DATA_BLOCK "InstProfinetDeviceDiag_x2"   // DB209
AUTHOR : Siemens Digital Industries
FAMILY : LAF
VERSION : 1.2
// stored: AssignedProDiagFB ProDiag, InstanceOfName LAF_ProfinetDevDiag, InstanceOfType FB
"LAF_ProfinetDevDiag"
   // VAR_INPUT
   //    plantIdentifier { ExternalAccessible := 'False'; ExternalVisible := 'False'; ExternalWritable := 'False'} : WString[24] := WSTRING#'';
   //    textListId { ExternalAccessible := 'False'; ExternalVisible := 'False'; ExternalWritable := 'False'} : Int := 0;
   //    localProfinetSystem { ExternalAccessible := 'False'; ExternalVisible := 'False'; ExternalWritable := 'False'} : HW_IOSYSTEM := 0;
   //    firstCycle { ExternalAccessible := 'False'; ExternalVisible := 'False'; ExternalWritable := 'False'} : Bool := FALSE;
   //    maxDevicesDiag { ExternalAccessible := 'False'; ExternalVisible := 'False'; ExternalWritable := 'False'} : DInt := 0;
   //    maxModulesDiag { ExternalAccessible := 'False'; ExternalVisible := 'False'; ExternalWritable := 'False'} : DInt := 0;
   //    ackAlarms { ExternalAccessible := 'False'; ExternalVisible := 'False'; ExternalWritable := 'False'} : Bool := FALSE;
   //    hideAlarmMask { ExternalAccessible := 'False'; ExternalVisible := 'False'; ExternalWritable := 'False'} : Word := 16#0000;
   // END_VAR
   // VAR_OUTPUT
   //    generalAlarm { ExternalAccessible := 'False'; ExternalVisible := 'False'; ExternalWritable := 'False'} : Bool := FALSE;
   //    deviceFaulty { ExternalAccessible := 'False'; ExternalVisible := 'False'; ExternalWritable := 'False'} : Bool := FALSE;
   //    deviceProblem { ExternalAccessible := 'False'; ExternalVisible := 'False'; ExternalWritable := 'False'} : Bool := FALSE;
   //    deviceDeactivated { ExternalAccessible := 'False'; ExternalVisible := 'False'; ExternalWritable := 'False'} : Bool := FALSE;
   //    deviceNotPresent { ExternalAccessible := 'False'; ExternalVisible := 'False'; ExternalWritable := 'False'} : Bool := FALSE;
   // END_VAR
   // VAR_IN_OUT
   //    interfaceDevDiag : "LAF_typeDevDiagInterface";
   // END_VAR
   // VAR
   //    statDevDiagInternal { ExternalAccessible := 'False'; ExternalVisible := 'False'; ExternalWritable := 'False'} : "LAF_typeDevDiagInternal";
   //    statCnt1ShotGetName { ExternalAccessible := 'False'; ExternalVisible := 'False'; ExternalWritable := 'False'} : DInt := 1;
   //    statCnt1ShotGeo2Log { ExternalAccessible := 'False'; ExternalVisible := 'False'; ExternalWritable := 'False'} : DInt := 1;
   //    statCnt1ShotGetImDat { ExternalAccessible := 'False'; ExternalVisible := 'False'; ExternalWritable := 'False'} : DInt := 1;
   //    statCntCyclDevState { ExternalAccessible := 'False'; ExternalVisible := 'False'; ExternalWritable := 'False'} : DInt := 1;
   //    statCntCyclState { ExternalAccessible := 'False'; ExternalVisible := 'False'; ExternalWritable := 'False'} : DInt := 1;
   //    statCntCyclModulState { ExternalAccessible := 'False'; ExternalVisible := 'False'; ExternalWritable := 'False'} : DInt := 1;
   //    statCntCyclGetDiag { ExternalAccessible := 'False'; ExternalVisible := 'False'; ExternalWritable := 'False'} : DInt := 1;
   //    statBusy { ExternalAccessible := 'False'; ExternalVisible := 'False'; ExternalWritable := 'False'} : "LAF_typeDevDiagStateInstruct";
   //    statDone { ExternalAccessible := 'False'; ExternalVisible := 'False'; ExternalWritable := 'False'} : "LAF_typeDevDiagStateInstruct";
   //    statOtherInstruct { ExternalAccessible := 'False'; ExternalVisible := 'False'; ExternalWritable := 'False'} : "LAF_typeDevDiagInstruct";
   //    instGetName { ExternalAccessible := 'False'; ExternalVisible := 'False'; ExternalWritable := 'False'} : Get_Name;
   //    statGetNameDat { ExternalAccessible := 'False'; ExternalVisible := 'False'; ExternalWritable := 'False'} : String[24] := '';
   //    statGetNameErrorStatus { ExternalAccessible := 'False'; ExternalVisible := 'False'; ExternalWritable := 'False'} : Word := 16#0000;
   //    statGetNameErrorDevCycle { ExternalAccessible := 'False'; ExternalVisible := 'False'; ExternalWritable := 'False'} : DInt := 0;
   //    instGetImData { ExternalAccessible := 'False'; ExternalVisible := 'False'; ExternalWritable := 'False'} : Get_IM_Data;
   //    statIm0Data { ExternalAccessible := 'False'; ExternalVisible := 'False'; ExternalWritable := 'False'} : IM0_Data;
   //    statGetImDatErrorStatus { ExternalAccessible := 'False'; ExternalVisible := 'False'; ExternalWritable := 'False'} : Word := 16#0000;
   //    statGetImDatErrorCycle { ExternalAccessible := 'False'; ExternalVisible := 'False'; ExternalWritable := 'False'} : DInt := 0;
   //    statAlarm { ExternalAccessible := 'False'; ExternalVisible := 'False'; ExternalWritable := 'False'} : "LAF_typeDevDiagAlarm";
   //    statHideAlarm { ExternalAccessible := 'False'; ExternalVisible := 'False'; ExternalWritable := 'False'} : "LAF_typeDevDiagAlarm";
   //    statRisPushbutton { ExternalAccessible := 'False'; ExternalVisible := 'False'; ExternalWritable := 'False'} : "LAF_typeDevDiagRisEdge";
   //    statErrorText { ExternalAccessible := 'False'; ExternalVisible := 'False'; ExternalWritable := 'False'} : String[24] := 'No Device Name readable';
   //    stat8CharError { ExternalAccessible := 'False'; ExternalVisible := 'False'; ExternalWritable := 'False'} : String[8] := '????????';
   //    statAlarmNo { ExternalAccessible := 'False'; ExternalVisible := 'False'; ExternalWritable := 'False'} : Array[0..23] of UInt;
   // END_VAR
BEGIN
   statDevDiagInternal.localProfinetSystem := 0;
   statDevDiagInternal.maxDevices := 0;
   statDevDiagInternal.maxModules := 0;
   statDevDiagInternal.numberDevices.configured := 0;
   statDevDiagInternal.numberDevices.notPresent := 0;
   statDevDiagInternal.numberDevices.deactivated := 0;
   statDevDiagInternal.numberDevices.faulty := 0;
   statDevDiagInternal.numberDevices.problem := 0;
   statDevDiagInternal.hwAddress[0..256].hwtype2 := 0;
   statDevDiagInternal.hwAddress[0..256].hwtype5 := 0;
   statDevDiagInternal.hwAddress[0..256].hwtype5If := 0;
   statBusy.getName := FALSE;
   statBusy.geo2Log := FALSE;
   statBusy.moduleStates := FALSE;
   statBusy.getDiag := FALSE;
   statBusy.getImData := FALSE;
   statDone.getName := FALSE;
   statDone.geo2Log := FALSE;
   statDone.moduleStates := FALSE;
   statDone.getDiag := FALSE;
   statDone.getImData := FALSE;
   statOtherInstruct.log2GeoLaddr := 0;
   statOtherInstruct.log2GeoRetVal := 0;
   statOtherInstruct.log2Geo.HWTYPE := 0;
   statOtherInstruct.log2Geo.AREA := 0;
   statOtherInstruct.log2Geo.IOSYSTEM := 0;
   statOtherInstruct.log2Geo.STATION := 0;
   statOtherInstruct.log2Geo.SLOT := 0;
   statOtherInstruct.log2Geo.SUBSLOT := 0;
   statOtherInstruct.devStateMode1.laddr := 0;
   statOtherInstruct.devStateMode1.mode := 0;
   statOtherInstruct.devStateMode1.retVal := 0;
   statOtherInstruct.devStateMode1.state[0..1024] := FALSE;
   statOtherInstruct.devStateMode2.laddr := 0;
   statOtherInstruct.devStateMode2.mode := 0;
   statOtherInstruct.devStateMode2.retVal := 0;
   statOtherInstruct.devStateMode2.state[0..1024] := FALSE;
   statOtherInstruct.devStateMode3.laddr := 0;
   statOtherInstruct.devStateMode3.mode := 0;
   statOtherInstruct.devStateMode3.retVal := 0;
   statOtherInstruct.devStateMode3.state[0..1024] := FALSE;
   statOtherInstruct.devStateMode4.laddr := 0;
   statOtherInstruct.devStateMode4.mode := 0;
   statOtherInstruct.devStateMode4.retVal := 0;
   statOtherInstruct.devStateMode4.state[0..1024] := FALSE;
   statOtherInstruct.devStateMode5.laddr := 0;
   statOtherInstruct.devStateMode5.mode := 0;
   statOtherInstruct.devStateMode5.retVal := 0;
   statOtherInstruct.devStateMode5.state[0..1024] := FALSE;
   statOtherInstruct.geo2LogLaddr := 0;
   statOtherInstruct.geo2LogRetVal := 0;
   statOtherInstruct.geo2Log.HWTYPE := 0;
   statOtherInstruct.geo2Log.AREA := 0;
   statOtherInstruct.geo2Log.IOSYSTEM := 0;
   statOtherInstruct.geo2Log.STATION := 0;
   statOtherInstruct.geo2Log.SLOT := 0;
   statOtherInstruct.geo2Log.SUBSLOT := 0;
   statOtherInstruct.moduleStateMode2.laddr := 0;
   statOtherInstruct.moduleStateMode2.mode := 0;
   statOtherInstruct.moduleStateMode2.retVal := 0;
   statOtherInstruct.moduleStateMode2.state[0..127] := FALSE;
   statOtherInstruct.moduleStateMode5.laddr := 0;
   statOtherInstruct.moduleStateMode5.mode := 0;
   statOtherInstruct.moduleStateMode5.retVal := 0;
   statOtherInstruct.moduleStateMode5.state[0..127] := FALSE;
   statOtherInstruct.getDiag.mode := 0;
   statOtherInstruct.getDiag.laddr := 0;
   statOtherInstruct.getDiag.retVal := 0;
   statOtherInstruct.getDiag.cntDiag := 0;
   statOtherInstruct.getDiag.diagDataMode0 := 16#0000_0000;
   statOtherInstruct.getDiag.diagDataMode1.MaintainanceState := 16#0000_0000;
   statOtherInstruct.getDiag.diagDataMode1.ComponentStateDetail := 16#0000_0000;
   statOtherInstruct.getDiag.diagDataMode1.OwnState := 0;
   statOtherInstruct.getDiag.diagDataMode1.IOState := 16#0000;
   statOtherInstruct.getDiag.diagDataMode1.OperatingState := 0;
   statOtherInstruct.getDiag.diagDataMode2.SubordinateState := 0;
   statOtherInstruct.getDiag.diagDataMode2.SubordinateIOState := 16#0000;
   statOtherInstruct.getDiag.diagDataMode2.DNNmode := 16#0000;
   statOtherInstruct.getDiag.detailData := 0;
   instGetName.LADDR := 0;
   instGetName.STATION_NR := 0;
   instGetName.DONE := FALSE;
   instGetName.BUSY := FALSE;
   instGetName.ERROR := FALSE;
   instGetName.LEN := 0;
   instGetName.STATUS := 16#0000;
   instGetName.BusyState := 16#0000;
   instGetImData.LADDR := 0;
   instGetImData.IM_TYPE := 0;
   instGetImData.DONE := FALSE;
   instGetImData.BUSY := FALSE;
   instGetImData.ERROR := FALSE;
   instGetImData.STATUS := 16#0000;
   instGetImData.sdw_GetAttrID := 16#0000_0000;
   instGetImData.sdw_GetAttrAID := 16#0000_0000;
   instGetImData.sdi_SfcLen := 0;
   instGetImData.sb_useGetMultiAttr := FALSE;
   instGetImData.sui_GetMultiAttrACount := 0;
   instGetImData.sa_GetMultiAttrPathLens[0] := 0;
   instGetImData.sa_GetMultiAttrPaths[0..2] := 0;
   instGetImData.sa_GetMultiAttrResultLens[0] := 0;
   instGetImData.sa_GetMultiAttrResult := '';
   instGetImData.sb_SfcValid := FALSE;
   instGetImData.sb_SfcERROR := FALSE;
   instGetImData.sw_SfcStatus := 16#0000;
   instGetImData.sa_SfcData[0..64] := 16#00;
   instGetImData.sudi_arraylength := 0;
   instGetImData.sudi_datatype := 0;
   instGetImData.sui_imdataLen := 0;
   instGetImData.sui_imdataLen_netto := 54;
   instGetImData.si_index := 0;
   instGetImData.sb_SfcLocked := FALSE;
   instGetImData.pw_TemporaryWord := 16#0000;
   instGetImData.pa_DataByte[0..53] := 16#00;
   instGetImData.pa_DataChar[0..53] := ' ';
   instGetImData.pa_TemporaryCharArray[0..19] := ' ';
   instGetImData.p_DataUDT.Manufacturer_ID := 0;
   instGetImData.p_DataUDT.Order_ID := '';
   instGetImData.p_DataUDT.Serial_Number := '';
   instGetImData.p_DataUDT.Hardware_Revision := 0;
   instGetImData.p_DataUDT.Software_Revision."Type" := ' ';
   instGetImData.p_DataUDT.Software_Revision.Functional := 0;
   instGetImData.p_DataUDT.Software_Revision.Bugfix := 0;
   instGetImData.p_DataUDT.Software_Revision.Internal := 0;
   instGetImData.p_DataUDT.Revision_Counter := 0;
   instGetImData.p_DataUDT.Profile_ID := 0;
   instGetImData.p_DataUDT.Profile_Specific_Type := 0;
   instGetImData.p_DataUDT.IM_Version := 16#0000;
   instGetImData.p_DataUDT.IM_Supported := 16#0000;
   statIm0Data.Manufacturer_ID := 0;
   statIm0Data.Order_ID := '';
   statIm0Data.Serial_Number := '';
   statIm0Data.Hardware_Revision := 0;
   statIm0Data.Software_Revision."Type" := ' ';
   statIm0Data.Software_Revision.Functional := 0;
   statIm0Data.Software_Revision.Bugfix := 0;
   statIm0Data.Software_Revision.Internal := 0;
   statIm0Data.Revision_Counter := 0;
   statIm0Data.Profile_ID := 0;
   statIm0Data.Profile_Specific_Type := 0;
   statIm0Data.IM_Version := 16#0000;
   statIm0Data.IM_Supported := 16#0000;
   statAlarm.invalidValueMaxDevices := FALSE;
   statAlarm.invalidValueMaxModules := FALSE;
   statAlarm.invalidAddressLog2Geo := FALSE;
   statAlarm.errorReadDeviceStates := FALSE;
   statAlarm.deviceFaulty := FALSE;
   statAlarm.deviceProblem := FALSE;
   statAlarm.deviceDeactivated := FALSE;
   statAlarm.deviceNotPresent := FALSE;
   statAlarm.deviceNetworkError := FALSE;
   statAlarm.deviceMaintRequired := FALSE;
   statAlarm.deviceMaintDemanded := FALSE;
   statAlarm.spare11 := FALSE;
   statAlarm.spare12 := FALSE;
   statAlarm.spare13 := FALSE;
   statAlarm.spare14 := FALSE;
   statAlarm.spare15 := FALSE;
   statHideAlarm.invalidValueMaxDevices := FALSE;
   statHideAlarm.invalidValueMaxModules := FALSE;
   statHideAlarm.invalidAddressLog2Geo := FALSE;
   statHideAlarm.errorReadDeviceStates := FALSE;
   statHideAlarm.deviceFaulty := FALSE;
   statHideAlarm.deviceProblem := FALSE;
   statHideAlarm.deviceDeactivated := FALSE;
   statHideAlarm.deviceNotPresent := FALSE;
   statHideAlarm.deviceNetworkError := FALSE;
   statHideAlarm.deviceMaintRequired := FALSE;
   statHideAlarm.deviceMaintDemanded := FALSE;
   statHideAlarm.spare11 := FALSE;
   statHideAlarm.spare12 := FALSE;
   statHideAlarm.spare13 := FALSE;
   statHideAlarm.spare14 := FALSE;
   statHideAlarm.spare15 := FALSE;
   statRisPushbutton.risEdgeManualReadAll := FALSE;
   statRisPushbutton.posPulseManualReadAll := FALSE;
   statRisPushbutton.risEdgeResetAll := FALSE;
   statRisPushbutton.posPulseResetAll := FALSE;
   statRisPushbutton.risEdgeQuitAlarms := FALSE;
   statRisPushbutton.posPulseQuitAlarms := FALSE;
   statAlarmNo[0] := 0;
   statAlarmNo[1] := 1;
   statAlarmNo[2] := 2;
   statAlarmNo[3] := 3;
   statAlarmNo[4] := 4;
   statAlarmNo[5] := 5;
   statAlarmNo[6] := 6;
   statAlarmNo[7] := 7;
   statAlarmNo[8] := 8;
   statAlarmNo[9] := 9;
   statAlarmNo[10] := 10;
   statAlarmNo[11] := 11;
   statAlarmNo[12] := 12;
   statAlarmNo[13] := 13;
   statAlarmNo[14] := 14;
   statAlarmNo[15] := 15;
   statAlarmNo[16] := 16;
   statAlarmNo[17] := 17;
   statAlarmNo[18] := 18;
   statAlarmNo[19] := 19;
   statAlarmNo[20] := 20;
   statAlarmNo[21] := 21;
   statAlarmNo[22] := 22;
   statAlarmNo[23] := 23;
END_DATA_BLOCK

DATA_BLOCK "CallInterfaceSignalsConv_BA10"   // DB347
// stored: InstanceOfName CallInterfaceSignalsConv, InstanceOfType FB
"CallInterfaceSignalsConv"
BEGIN
   signalsS2R.Load_Enable := FALSE;
   signalsS2R.Load_Complete_Comfirm := FALSE;
   signalsS2R.Cell_Data_Report := FALSE;
   signalsS2R.signal3 := FALSE;
   signalsS2R.signal4 := FALSE;
   signalsS2R.signal5 := FALSE;
   signalsS2R.signal6 := FALSE;
   signalsS2R.signal7 := FALSE;
   signalsS2R.signal8 := FALSE;
   signalsS2R.signal9 := FALSE;
   signalsS2R.signal10 := FALSE;
   signalsS2R.signal11 := FALSE;
   signalsS2R.signal12 := FALSE;
   signalsS2R.signal13 := FALSE;
   signalsS2R.signal14 := FALSE;
   signalsS2R.HeartBeat := FALSE;
   signalsS2R.signal16 := FALSE;
   signalsS2R.signal17 := FALSE;
   signalsS2R.signal18 := FALSE;
   signalsS2R.signal19 := FALSE;
   signalsS2R.signal20 := FALSE;
   signalsS2R.signal21 := FALSE;
   signalsS2R.signal22 := FALSE;
   signalsS2R.signal23 := FALSE;
   signalsS2R.signal24 := FALSE;
   signalsS2R.signal25 := FALSE;
   signalsS2R.signal26 := FALSE;
   signalsS2R.signal27 := FALSE;
   signalsS2R.signal28 := FALSE;
   signalsS2R.signal29 := FALSE;
   signalsS2R.signal30 := FALSE;
   signalsS2R.signal31 := FALSE;
   signalsS2R.signal32 := FALSE;
   signalsS2R.signal33 := FALSE;
   signalsS2R.signal34 := FALSE;
   signalsS2R.signal35 := FALSE;
   signalsS2R.signal36 := FALSE;
   signalsS2R.signal37 := FALSE;
   signalsS2R.signal38 := FALSE;
   signalsS2R.signal39 := FALSE;
   signalsS2R.signal40 := FALSE;
   signalsS2R.signal41 := FALSE;
   signalsS2R.signal42 := FALSE;
   signalsS2R.signal43 := FALSE;
   signalsS2R.signal44 := FALSE;
   signalsS2R.signal45 := FALSE;
   signalsS2R.signal46 := FALSE;
   signalsS2R.signal47 := FALSE;
   signalsS2R.signal48 := FALSE;
   signalsS2R.signal49 := FALSE;
   signalsS2R.signal50 := FALSE;
   signalsS2R.signal51 := FALSE;
   signalsS2R.signal52 := FALSE;
   signalsS2R.signal53 := FALSE;
   signalsS2R.signal54 := FALSE;
   signalsS2R.signal55 := FALSE;
   signalsS2R.signal56 := FALSE;
   signalsS2R.signal57 := FALSE;
   signalsS2R.signal58 := FALSE;
   signalsS2R.signal59 := FALSE;
   signalsS2R.signal60 := FALSE;
   signalsS2R.signal61 := FALSE;
   signalsS2R.signal62 := FALSE;
   signalsS2R.signal63 := FALSE;
   signalsS2R.signal64 := FALSE;
   signalsS2R.signal65 := FALSE;
   signalsS2R.signal66 := FALSE;
   signalsS2R.signal67 := FALSE;
   signalsS2R.signal68 := FALSE;
   signalsS2R.signal69 := FALSE;
   signalsS2R.signal70 := FALSE;
   signalsS2R.signal71 := FALSE;
   signalsS2R.signal72 := FALSE;
   signalsS2R.signal73 := FALSE;
   signalsS2R.signal74 := FALSE;
   signalsS2R.signal75 := FALSE;
   signalsS2R.signal76 := FALSE;
   signalsS2R.signal77 := FALSE;
   signalsS2R.signal78 := FALSE;
   signalsS2R.signal79 := FALSE;
   signalsS2R.signal80 := FALSE;
   signalsS2R.signal81 := FALSE;
   signalsS2R.signal82 := FALSE;
   signalsS2R.signal83 := FALSE;
   signalsS2R.signal84 := FALSE;
   signalsS2R.signal85 := FALSE;
   signalsS2R.signal86 := FALSE;
   signalsS2R.signal87 := FALSE;
   signalsS2R.signal88 := FALSE;
   signalsS2R.signal89 := FALSE;
   signalsS2R.signal90 := FALSE;
   signalsS2R.signal91 := FALSE;
   signalsS2R.signal92 := FALSE;
   signalsS2R.signal93 := FALSE;
   signalsS2R.signal94 := FALSE;
   signalsS2R.signal95 := FALSE;
   signalsR2S.Load_Requset := FALSE;
   signalsR2S.Load_Busy := FALSE;
   signalsR2S.Load_Complete := FALSE;
   signalsR2S.Cell_Data_Request := FALSE;
   signalsR2S.Cell_Data_Report_Ack := FALSE;
   signalsR2S.Cell_Data_Report_Nck := FALSE;
   signalsR2S.signal6 := FALSE;
   signalsR2S.signal7 := FALSE;
   signalsR2S.signal8 := FALSE;
   signalsR2S.signal9 := FALSE;
   signalsR2S.signal10 := FALSE;
   signalsR2S.signal11 := FALSE;
   signalsR2S.signal12 := FALSE;
   signalsR2S.signal13 := FALSE;
   signalsR2S.signal14 := FALSE;
   signalsR2S.HeartBeat := FALSE;
   signalsR2S.signal16 := FALSE;
   signalsR2S.signal17 := FALSE;
   signalsR2S.signal18 := FALSE;
   signalsR2S.signal19 := FALSE;
   signalsR2S.signal20 := FALSE;
   signalsR2S.signal21 := FALSE;
   signalsR2S.signal22 := FALSE;
   signalsR2S.signal23 := FALSE;
   signalsR2S.signal24 := FALSE;
   signalsR2S.signal25 := FALSE;
   signalsR2S.signal26 := FALSE;
   signalsR2S.signal27 := FALSE;
   signalsR2S.signal28 := FALSE;
   signalsR2S.signal29 := FALSE;
   signalsR2S.signal30 := FALSE;
   signalsR2S.signal31 := FALSE;
   signalsR2S.signal32 := FALSE;
   signalsR2S.signal33 := FALSE;
   signalsR2S.signal34 := FALSE;
   signalsR2S.signal35 := FALSE;
   signalsR2S.signal36 := FALSE;
   signalsR2S.signal37 := FALSE;
   signalsR2S.signal38 := FALSE;
   signalsR2S.signal39 := FALSE;
   signalsR2S.signal40 := FALSE;
   signalsR2S.signal41 := FALSE;
   signalsR2S.signal42 := FALSE;
   signalsR2S.signal43 := FALSE;
   signalsR2S.signal44 := FALSE;
   signalsR2S.signal45 := FALSE;
   signalsR2S.signal46 := FALSE;
   signalsR2S.signal47 := FALSE;
   signalsR2S.signal48 := FALSE;
   signalsR2S.signal49 := FALSE;
   signalsR2S.signal50 := FALSE;
   signalsR2S.signal51 := FALSE;
   signalsR2S.signal52 := FALSE;
   signalsR2S.signal53 := FALSE;
   signalsR2S.signal54 := FALSE;
   signalsR2S.signal55 := FALSE;
   signalsR2S.signal56 := FALSE;
   signalsR2S.signal57 := FALSE;
   signalsR2S.signal58 := FALSE;
   signalsR2S.signal59 := FALSE;
   signalsR2S.signal60 := FALSE;
   signalsR2S.signal61 := FALSE;
   signalsR2S.signal62 := FALSE;
   signalsR2S.signal63 := FALSE;
   signalsR2S.signal64 := FALSE;
   signalsR2S.signal65 := FALSE;
   signalsR2S.signal66 := FALSE;
   signalsR2S.signal67 := FALSE;
   signalsR2S.signal68 := FALSE;
   signalsR2S.signal69 := FALSE;
   signalsR2S.signal70 := FALSE;
   signalsR2S.signal71 := FALSE;
   signalsR2S.signal72 := FALSE;
   signalsR2S.signal73 := FALSE;
   signalsR2S.signal74 := FALSE;
   signalsR2S.signal75 := FALSE;
   signalsR2S.signal76 := FALSE;
   signalsR2S.signal77 := FALSE;
   signalsR2S.signal78 := FALSE;
   signalsR2S.signal79 := FALSE;
   signalsR2S.signal80 := FALSE;
   signalsR2S.signal81 := FALSE;
   signalsR2S.signal82 := FALSE;
   signalsR2S.signal83 := FALSE;
   signalsR2S.signal84 := FALSE;
   signalsR2S.signal85 := FALSE;
   signalsR2S.signal86 := FALSE;
   signalsR2S.signal87 := FALSE;
   signalsR2S.signal88 := FALSE;
   signalsR2S.signal89 := FALSE;
   signalsR2S.signal90 := FALSE;
   signalsR2S.signal91 := FALSE;
   signalsR2S.signal92 := FALSE;
   signalsR2S.signal93 := FALSE;
   signalsR2S.signal94 := FALSE;
   signalsR2S.signal95 := FALSE;
   statWordBuffer_2[0..5] := 16#0000;
   statWordBuffer_1[0..5] := 16#0000;
END_DATA_BLOCK

DATA_BLOCK "CallInterfaceSignalsConv_BA15"   // DB348
// stored: InstanceOfName CallInterfaceSignalsConv, InstanceOfType FB
"CallInterfaceSignalsConv"
BEGIN
   signalsS2R.Load_Enable := FALSE;
   signalsS2R.Load_Complete_Comfirm := FALSE;
   signalsS2R.Cell_Data_Report := FALSE;
   signalsS2R.signal3 := FALSE;
   signalsS2R.signal4 := FALSE;
   signalsS2R.signal5 := FALSE;
   signalsS2R.signal6 := FALSE;
   signalsS2R.signal7 := FALSE;
   signalsS2R.signal8 := FALSE;
   signalsS2R.signal9 := FALSE;
   signalsS2R.signal10 := FALSE;
   signalsS2R.signal11 := FALSE;
   signalsS2R.signal12 := FALSE;
   signalsS2R.signal13 := FALSE;
   signalsS2R.signal14 := FALSE;
   signalsS2R.HeartBeat := FALSE;
   signalsS2R.signal16 := FALSE;
   signalsS2R.signal17 := FALSE;
   signalsS2R.signal18 := FALSE;
   signalsS2R.signal19 := FALSE;
   signalsS2R.signal20 := FALSE;
   signalsS2R.signal21 := FALSE;
   signalsS2R.signal22 := FALSE;
   signalsS2R.signal23 := FALSE;
   signalsS2R.signal24 := FALSE;
   signalsS2R.signal25 := FALSE;
   signalsS2R.signal26 := FALSE;
   signalsS2R.signal27 := FALSE;
   signalsS2R.signal28 := FALSE;
   signalsS2R.signal29 := FALSE;
   signalsS2R.signal30 := FALSE;
   signalsS2R.signal31 := FALSE;
   signalsS2R.signal32 := FALSE;
   signalsS2R.signal33 := FALSE;
   signalsS2R.signal34 := FALSE;
   signalsS2R.signal35 := FALSE;
   signalsS2R.signal36 := FALSE;
   signalsS2R.signal37 := FALSE;
   signalsS2R.signal38 := FALSE;
   signalsS2R.signal39 := FALSE;
   signalsS2R.signal40 := FALSE;
   signalsS2R.signal41 := FALSE;
   signalsS2R.signal42 := FALSE;
   signalsS2R.signal43 := FALSE;
   signalsS2R.signal44 := FALSE;
   signalsS2R.signal45 := FALSE;
   signalsS2R.signal46 := FALSE;
   signalsS2R.signal47 := FALSE;
   signalsS2R.signal48 := FALSE;
   signalsS2R.signal49 := FALSE;
   signalsS2R.signal50 := FALSE;
   signalsS2R.signal51 := FALSE;
   signalsS2R.signal52 := FALSE;
   signalsS2R.signal53 := FALSE;
   signalsS2R.signal54 := FALSE;
   signalsS2R.signal55 := FALSE;
   signalsS2R.signal56 := FALSE;
   signalsS2R.signal57 := FALSE;
   signalsS2R.signal58 := FALSE;
   signalsS2R.signal59 := FALSE;
   signalsS2R.signal60 := FALSE;
   signalsS2R.signal61 := FALSE;
   signalsS2R.signal62 := FALSE;
   signalsS2R.signal63 := FALSE;
   signalsS2R.signal64 := FALSE;
   signalsS2R.signal65 := FALSE;
   signalsS2R.signal66 := FALSE;
   signalsS2R.signal67 := FALSE;
   signalsS2R.signal68 := FALSE;
   signalsS2R.signal69 := FALSE;
   signalsS2R.signal70 := FALSE;
   signalsS2R.signal71 := FALSE;
   signalsS2R.signal72 := FALSE;
   signalsS2R.signal73 := FALSE;
   signalsS2R.signal74 := FALSE;
   signalsS2R.signal75 := FALSE;
   signalsS2R.signal76 := FALSE;
   signalsS2R.signal77 := FALSE;
   signalsS2R.signal78 := FALSE;
   signalsS2R.signal79 := FALSE;
   signalsS2R.signal80 := FALSE;
   signalsS2R.signal81 := FALSE;
   signalsS2R.signal82 := FALSE;
   signalsS2R.signal83 := FALSE;
   signalsS2R.signal84 := FALSE;
   signalsS2R.signal85 := FALSE;
   signalsS2R.signal86 := FALSE;
   signalsS2R.signal87 := FALSE;
   signalsS2R.signal88 := FALSE;
   signalsS2R.signal89 := FALSE;
   signalsS2R.signal90 := FALSE;
   signalsS2R.signal91 := FALSE;
   signalsS2R.signal92 := FALSE;
   signalsS2R.signal93 := FALSE;
   signalsS2R.signal94 := FALSE;
   signalsS2R.signal95 := FALSE;
   signalsR2S.Load_Requset := FALSE;
   signalsR2S.Load_Busy := FALSE;
   signalsR2S.Load_Complete := FALSE;
   signalsR2S.Cell_Data_Request := FALSE;
   signalsR2S.Cell_Data_Report_Ack := FALSE;
   signalsR2S.Cell_Data_Report_Nck := FALSE;
   signalsR2S.signal6 := FALSE;
   signalsR2S.signal7 := FALSE;
   signalsR2S.signal8 := FALSE;
   signalsR2S.signal9 := FALSE;
   signalsR2S.signal10 := FALSE;
   signalsR2S.signal11 := FALSE;
   signalsR2S.signal12 := FALSE;
   signalsR2S.signal13 := FALSE;
   signalsR2S.signal14 := FALSE;
   signalsR2S.HeartBeat := FALSE;
   signalsR2S.signal16 := FALSE;
   signalsR2S.signal17 := FALSE;
   signalsR2S.signal18 := FALSE;
   signalsR2S.signal19 := FALSE;
   signalsR2S.signal20 := FALSE;
   signalsR2S.signal21 := FALSE;
   signalsR2S.signal22 := FALSE;
   signalsR2S.signal23 := FALSE;
   signalsR2S.signal24 := FALSE;
   signalsR2S.signal25 := FALSE;
   signalsR2S.signal26 := FALSE;
   signalsR2S.signal27 := FALSE;
   signalsR2S.signal28 := FALSE;
   signalsR2S.signal29 := FALSE;
   signalsR2S.signal30 := FALSE;
   signalsR2S.signal31 := FALSE;
   signalsR2S.signal32 := FALSE;
   signalsR2S.signal33 := FALSE;
   signalsR2S.signal34 := FALSE;
   signalsR2S.signal35 := FALSE;
   signalsR2S.signal36 := FALSE;
   signalsR2S.signal37 := FALSE;
   signalsR2S.signal38 := FALSE;
   signalsR2S.signal39 := FALSE;
   signalsR2S.signal40 := FALSE;
   signalsR2S.signal41 := FALSE;
   signalsR2S.signal42 := FALSE;
   signalsR2S.signal43 := FALSE;
   signalsR2S.signal44 := FALSE;
   signalsR2S.signal45 := FALSE;
   signalsR2S.signal46 := FALSE;
   signalsR2S.signal47 := FALSE;
   signalsR2S.signal48 := FALSE;
   signalsR2S.signal49 := FALSE;
   signalsR2S.signal50 := FALSE;
   signalsR2S.signal51 := FALSE;
   signalsR2S.signal52 := FALSE;
   signalsR2S.signal53 := FALSE;
   signalsR2S.signal54 := FALSE;
   signalsR2S.signal55 := FALSE;
   signalsR2S.signal56 := FALSE;
   signalsR2S.signal57 := FALSE;
   signalsR2S.signal58 := FALSE;
   signalsR2S.signal59 := FALSE;
   signalsR2S.signal60 := FALSE;
   signalsR2S.signal61 := FALSE;
   signalsR2S.signal62 := FALSE;
   signalsR2S.signal63 := FALSE;
   signalsR2S.signal64 := FALSE;
   signalsR2S.signal65 := FALSE;
   signalsR2S.signal66 := FALSE;
   signalsR2S.signal67 := FALSE;
   signalsR2S.signal68 := FALSE;
   signalsR2S.signal69 := FALSE;
   signalsR2S.signal70 := FALSE;
   signalsR2S.signal71 := FALSE;
   signalsR2S.signal72 := FALSE;
   signalsR2S.signal73 := FALSE;
   signalsR2S.signal74 := FALSE;
   signalsR2S.signal75 := FALSE;
   signalsR2S.signal76 := FALSE;
   signalsR2S.signal77 := FALSE;
   signalsR2S.signal78 := FALSE;
   signalsR2S.signal79 := FALSE;
   signalsR2S.signal80 := FALSE;
   signalsR2S.signal81 := FALSE;
   signalsR2S.signal82 := FALSE;
   signalsR2S.signal83 := FALSE;
   signalsR2S.signal84 := FALSE;
   signalsR2S.signal85 := FALSE;
   signalsR2S.signal86 := FALSE;
   signalsR2S.signal87 := FALSE;
   signalsR2S.signal88 := FALSE;
   signalsR2S.signal89 := FALSE;
   signalsR2S.signal90 := FALSE;
   signalsR2S.signal91 := FALSE;
   signalsR2S.signal92 := FALSE;
   signalsR2S.signal93 := FALSE;
   signalsR2S.signal94 := FALSE;
   signalsR2S.signal95 := FALSE;
   statWordBuffer_2[0..5] := 16#0000;
   statWordBuffer_1[0..5] := 16#0000;
END_DATA_BLOCK

DATA_BLOCK "InterfaceSignals"   // DB232
// stored: Access Published, InstanceOfName LER_SignalsInterface, InstanceOfType UDT
"LER_SignalsInterface"
   // VAR
   //    HMI_Select_Mode : Bool := FALSE;
   //    ButtonValue : Array[0..16] of "LER_SignalsInput";
   // END_VAR
BEGIN
   ButtonValue[0].ButtonLeft[0..15] := FALSE;
   ButtonValue[1].ButtonLeft[0..15] := FALSE;
   ButtonValue[2].ButtonLeft[0..15] := FALSE;
   ButtonValue[3].ButtonLeft[0..15] := FALSE;
   ButtonValue[4].ButtonLeft[0..15] := FALSE;
   ButtonValue[5].ButtonLeft[0..15] := FALSE;
   ButtonValue[6].ButtonLeft[0..15] := FALSE;
   ButtonValue[7].ButtonLeft[0..15] := FALSE;
   ButtonValue[8].ButtonLeft[0..15] := FALSE;
   ButtonValue[9].ButtonLeft[0..15] := FALSE;
   ButtonValue[10].ButtonLeft[0..15] := FALSE;
   ButtonValue[11].ButtonLeft[0..15] := FALSE;
   ButtonValue[12].ButtonLeft[0..15] := FALSE;
   ButtonValue[13].ButtonLeft[0..15] := FALSE;
   ButtonValue[14].ButtonLeft[0..15] := FALSE;
   ButtonValue[15].ButtonLeft[0..15] := FALSE;
   ButtonValue[16].ButtonLeft[0..15] := FALSE;
   ButtonValue[0].ButtonRight[0..15] := FALSE;
   ButtonValue[1].ButtonRight[0..15] := FALSE;
   ButtonValue[2].ButtonRight[0..15] := FALSE;
   ButtonValue[3].ButtonRight[0..15] := FALSE;
   ButtonValue[4].ButtonRight[0..15] := FALSE;
   ButtonValue[5].ButtonRight[0..15] := FALSE;
   ButtonValue[6].ButtonRight[0..15] := FALSE;
   ButtonValue[7].ButtonRight[0..15] := FALSE;
   ButtonValue[8].ButtonRight[0..15] := FALSE;
   ButtonValue[9].ButtonRight[0..15] := FALSE;
   ButtonValue[10].ButtonRight[0..15] := FALSE;
   ButtonValue[11].ButtonRight[0..15] := FALSE;
   ButtonValue[12].ButtonRight[0..15] := FALSE;
   ButtonValue[13].ButtonRight[0..15] := FALSE;
   ButtonValue[14].ButtonRight[0..15] := FALSE;
   ButtonValue[15].ButtonRight[0..15] := FALSE;
   ButtonValue[16].ButtonRight[0..15] := FALSE;
END_DATA_BLOCK

DATA_BLOCK "ReelCutToStack10"   // DB329
// stored: InstanceOfName typeReelCutToStack, InstanceOfType UDT
"typeReelCutToStack"
BEGIN
END_DATA_BLOCK

DATA_BLOCK "ReelCutToStack15"   // DB330
// stored: InstanceOfName typeReelCutToStack, InstanceOfType UDT
"typeReelCutToStack"
BEGIN
END_DATA_BLOCK

DATA_BLOCK "StackToReelCut10"   // DB331
// stored: InstanceOfName typeStackToReelCut, InstanceOfType UDT
"typeStackToReelCut"
BEGIN
END_DATA_BLOCK

DATA_BLOCK "StackToReelCut15"   // DB332
// stored: InstanceOfName typeStackToReelCut, InstanceOfType UDT
"typeStackToReelCut"
BEGIN
END_DATA_BLOCK

DATA_BLOCK "instGetMotorstarterSignals"   // DB91
// stored: InstanceOfName GetMotorstarterSignals, InstanceOfType FB
"GetMotorstarterSignals"
BEGIN
   Et200SpMotorstarterInterfaceAllUnits[0].EMmotorstarter[0].et200SpMotorstarterCurrent[0..1] := 0.0;
   Et200SpMotorstarterInterfaceAllUnits[0].EMmotorstarter[1].et200SpMotorstarterCurrent[0..1] := 0.0;
   Et200SpMotorstarterInterfaceAllUnits[0].EMmotorstarter[2].et200SpMotorstarterCurrent[0..1] := 0.0;
   Et200SpMotorstarterInterfaceAllUnits[0].EMmotorstarter[3].et200SpMotorstarterCurrent[0..1] := 0.0;
   Et200SpMotorstarterInterfaceAllUnits[0].EMmotorstarter[4].et200SpMotorstarterCurrent[0..1] := 0.0;
   Et200SpMotorstarterInterfaceAllUnits[0].EMmotorstarter[5].et200SpMotorstarterCurrent[0..1] := 0.0;
   Et200SpMotorstarterInterfaceAllUnits[0].EMmotorstarter[6].et200SpMotorstarterCurrent[0..1] := 0.0;
   Et200SpMotorstarterInterfaceAllUnits[0].EMmotorstarter[7].et200SpMotorstarterCurrent[0..1] := 0.0;
   Et200SpMotorstarterInterfaceAllUnits[0].EMmotorstarter[0].et200SpMotorstarterInputs[0..1].readyAutomatic := FALSE;
   Et200SpMotorstarterInterfaceAllUnits[0].EMmotorstarter[1].et200SpMotorstarterInputs[0..1].readyAutomatic := FALSE;
   Et200SpMotorstarterInterfaceAllUnits[0].EMmotorstarter[2].et200SpMotorstarterInputs[0..1].readyAutomatic := FALSE;
   Et200SpMotorstarterInterfaceAllUnits[0].EMmotorstarter[3].et200SpMotorstarterInputs[0..1].readyAutomatic := FALSE;
   Et200SpMotorstarterInterfaceAllUnits[0].EMmotorstarter[4].et200SpMotorstarterInputs[0..1].readyAutomatic := FALSE;
   Et200SpMotorstarterInterfaceAllUnits[0].EMmotorstarter[5].et200SpMotorstarterInputs[0..1].readyAutomatic := FALSE;
   Et200SpMotorstarterInterfaceAllUnits[0].EMmotorstarter[6].et200SpMotorstarterInputs[0..1].readyAutomatic := FALSE;
   Et200SpMotorstarterInterfaceAllUnits[0].EMmotorstarter[7].et200SpMotorstarterInputs[0..1].readyAutomatic := FALSE;
   Et200SpMotorstarterInterfaceAllUnits[0].EMmotorstarter[0].et200SpMotorstarterInputs[0..1].motorOn := FALSE;
   Et200SpMotorstarterInterfaceAllUnits[0].EMmotorstarter[1].et200SpMotorstarterInputs[0..1].motorOn := FALSE;
   Et200SpMotorstarterInterfaceAllUnits[0].EMmotorstarter[2].et200SpMotorstarterInputs[0..1].motorOn := FALSE;
   Et200SpMotorstarterInterfaceAllUnits[0].EMmotorstarter[3].et200SpMotorstarterInputs[0..1].motorOn := FALSE;
   Et200SpMotorstarterInterfaceAllUnits[0].EMmotorstarter[4].et200SpMotorstarterInputs[0..1].motorOn := FALSE;
   Et200SpMotorstarterInterfaceAllUnits[0].EMmotorstarter[5].et200SpMotorstarterInputs[0..1].motorOn := FALSE;
   Et200SpMotorstarterInterfaceAllUnits[0].EMmotorstarter[6].et200SpMotorstarterInputs[0..1].motorOn := FALSE;
   Et200SpMotorstarterInterfaceAllUnits[0].EMmotorstarter[7].et200SpMotorstarterInputs[0..1].motorOn := FALSE;
   Et200SpMotorstarterInterfaceAllUnits[0].EMmotorstarter[0].et200SpMotorstarterInputs[0..1].groupFault := FALSE;
   Et200SpMotorstarterInterfaceAllUnits[0].EMmotorstarter[1].et200SpMotorstarterInputs[0..1].groupFault := FALSE;
   Et200SpMotorstarterInterfaceAllUnits[0].EMmotorstarter[2].et200SpMotorstarterInputs[0..1].groupFault := FALSE;
   Et200SpMotorstarterInterfaceAllUnits[0].EMmotorstarter[3].et200SpMotorstarterInputs[0..1].groupFault := FALSE;
   Et200SpMotorstarterInterfaceAllUnits[0].EMmotorstarter[4].et200SpMotorstarterInputs[0..1].groupFault := FALSE;
   Et200SpMotorstarterInterfaceAllUnits[0].EMmotorstarter[5].et200SpMotorstarterInputs[0..1].groupFault := FALSE;
   Et200SpMotorstarterInterfaceAllUnits[0].EMmotorstarter[6].et200SpMotorstarterInputs[0..1].groupFault := FALSE;
   Et200SpMotorstarterInterfaceAllUnits[0].EMmotorstarter[7].et200SpMotorstarterInputs[0..1].groupFault := FALSE;
   Et200SpMotorstarterInterfaceAllUnits[0].EMmotorstarter[0].et200SpMotorstarterInputs[0..1].groupWarning := FALSE;
   Et200SpMotorstarterInterfaceAllUnits[0].EMmotorstarter[1].et200SpMotorstarterInputs[0..1].groupWarning := FALSE;
   Et200SpMotorstarterInterfaceAllUnits[0].EMmotorstarter[2].et200SpMotorstarterInputs[0..1].groupWarning := FALSE;
   Et200SpMotorstarterInterfaceAllUnits[0].EMmotorstarter[3].et200SpMotorstarterInputs[0..1].groupWarning := FALSE;
   Et200SpMotorstarterInterfaceAllUnits[0].EMmotorstarter[4].et200SpMotorstarterInputs[0..1].groupWarning := FALSE;
   Et200SpMotorstarterInterfaceAllUnits[0].EMmotorstarter[5].et200SpMotorstarterInputs[0..1].groupWarning := FALSE;
   Et200SpMotorstarterInterfaceAllUnits[0].EMmotorstarter[6].et200SpMotorstarterInputs[0..1].groupWarning := FALSE;
   Et200SpMotorstarterInterfaceAllUnits[0].EMmotorstarter[7].et200SpMotorstarterInputs[0..1].groupWarning := FALSE;
   Et200SpMotorstarterInterfaceAllUnits[0].EMmotorstarter[0].et200SpMotorstarterInputs[0..1].input1 := FALSE;
   Et200SpMotorstarterInterfaceAllUnits[0].EMmotorstarter[1].et200SpMotorstarterInputs[0..1].input1 := FALSE;
   Et200SpMotorstarterInterfaceAllUnits[0].EMmotorstarter[2].et200SpMotorstarterInputs[0..1].input1 := FALSE;
   Et200SpMotorstarterInterfaceAllUnits[0].EMmotorstarter[3].et200SpMotorstarterInputs[0..1].input1 := FALSE;
   Et200SpMotorstarterInterfaceAllUnits[0].EMmotorstarter[4].et200SpMotorstarterInputs[0..1].input1 := FALSE;
   Et200SpMotorstarterInterfaceAllUnits[0].EMmotorstarter[5].et200SpMotorstarterInputs[0..1].input1 := FALSE;
   Et200SpMotorstarterInterfaceAllUnits[0].EMmotorstarter[6].et200SpMotorstarterInputs[0..1].input1 := FALSE;
   Et200SpMotorstarterInterfaceAllUnits[0].EMmotorstarter[7].et200SpMotorstarterInputs[0..1].input1 := FALSE;
   Et200SpMotorstarterInterfaceAllUnits[0].EMmotorstarter[0].et200SpMotorstarterInputs[0..1].input2 := FALSE;
   Et200SpMotorstarterInterfaceAllUnits[0].EMmotorstarter[1].et200SpMotorstarterInputs[0..1].input2 := FALSE;
   Et200SpMotorstarterInterfaceAllUnits[0].EMmotorstarter[2].et200SpMotorstarterInputs[0..1].input2 := FALSE;
   Et200SpMotorstarterInterfaceAllUnits[0].EMmotorstarter[3].et200SpMotorstarterInputs[0..1].input2 := FALSE;
   Et200SpMotorstarterInterfaceAllUnits[0].EMmotorstarter[4].et200SpMotorstarterInputs[0..1].input2 := FALSE;
   Et200SpMotorstarterInterfaceAllUnits[0].EMmotorstarter[5].et200SpMotorstarterInputs[0..1].input2 := FALSE;
   Et200SpMotorstarterInterfaceAllUnits[0].EMmotorstarter[6].et200SpMotorstarterInputs[0..1].input2 := FALSE;
   Et200SpMotorstarterInterfaceAllUnits[0].EMmotorstarter[7].et200SpMotorstarterInputs[0..1].input2 := FALSE;
   Et200SpMotorstarterInterfaceAllUnits[0].EMmotorstarter[0].et200SpMotorstarterInputs[0..1].input3 := FALSE;
   Et200SpMotorstarterInterfaceAllUnits[0].EMmotorstarter[1].et200SpMotorstarterInputs[0..1].input3 := FALSE;
   Et200SpMotorstarterInterfaceAllUnits[0].EMmotorstarter[2].et200SpMotorstarterInputs[0..1].input3 := FALSE;
   Et200SpMotorstarterInterfaceAllUnits[0].EMmotorstarter[3].et200SpMotorstarterInputs[0..1].input3 := FALSE;
   Et200SpMotorstarterInterfaceAllUnits[0].EMmotorstarter[4].et200SpMotorstarterInputs[0..1].input3 := FALSE;
   Et200SpMotorstarterInterfaceAllUnits[0].EMmotorstarter[5].et200SpMotorstarterInputs[0..1].input3 := FALSE;
   Et200SpMotorstarterInterfaceAllUnits[0].EMmotorstarter[6].et200SpMotorstarterInputs[0..1].input3 := FALSE;
   Et200SpMotorstarterInterfaceAllUnits[0].EMmotorstarter[7].et200SpMotorstarterInputs[0..1].input3 := FALSE;
   Et200SpMotorstarterInterfaceAllUnits[0].EMmotorstarter[0].et200SpMotorstarterInputs[0..1].inputLocalCtrl := FALSE;
   Et200SpMotorstarterInterfaceAllUnits[0].EMmotorstarter[1].et200SpMotorstarterInputs[0..1].inputLocalCtrl := FALSE;
   Et200SpMotorstarterInterfaceAllUnits[0].EMmotorstarter[2].et200SpMotorstarterInputs[0..1].inputLocalCtrl := FALSE;
   Et200SpMotorstarterInterfaceAllUnits[0].EMmotorstarter[3].et200SpMotorstarterInputs[0..1].inputLocalCtrl := FALSE;
   Et200SpMotorstarterInterfaceAllUnits[0].EMmotorstarter[4].et200SpMotorstarterInputs[0..1].inputLocalCtrl := FALSE;
   Et200SpMotorstarterInterfaceAllUnits[0].EMmotorstarter[5].et200SpMotorstarterInputs[0..1].inputLocalCtrl := FALSE;
   Et200SpMotorstarterInterfaceAllUnits[0].EMmotorstarter[6].et200SpMotorstarterInputs[0..1].inputLocalCtrl := FALSE;
   Et200SpMotorstarterInterfaceAllUnits[0].EMmotorstarter[7].et200SpMotorstarterInputs[0..1].inputLocalCtrl := FALSE;
   Et200SpMotorstarterInterfaceAllUnits[0].EMmotorstarter[0].et200SpMotorstarterInputs[0..1].iActBit0 := FALSE;
   Et200SpMotorstarterInterfaceAllUnits[0].EMmotorstarter[1].et200SpMotorstarterInputs[0..1].iActBit0 := FALSE;
   Et200SpMotorstarterInterfaceAllUnits[0].EMmotorstarter[2].et200SpMotorstarterInputs[0..1].iActBit0 := FALSE;
   Et200SpMotorstarterInterfaceAllUnits[0].EMmotorstarter[3].et200SpMotorstarterInputs[0..1].iActBit0 := FALSE;
   Et200SpMotorstarterInterfaceAllUnits[0].EMmotorstarter[4].et200SpMotorstarterInputs[0..1].iActBit0 := FALSE;
   Et200SpMotorstarterInterfaceAllUnits[0].EMmotorstarter[5].et200SpMotorstarterInputs[0..1].iActBit0 := FALSE;
   Et200SpMotorstarterInterfaceAllUnits[0].EMmotorstarter[6].et200SpMotorstarterInputs[0..1].iActBit0 := FALSE;
   Et200SpMotorstarterInterfaceAllUnits[0].EMmotorstarter[7].et200SpMotorstarterInputs[0..1].iActBit0 := FALSE;
   Et200SpMotorstarterInterfaceAllUnits[0].EMmotorstarter[0].et200SpMotorstarterInputs[0..1].iActBit1 := FALSE;
   Et200SpMotorstarterInterfaceAllUnits[0].EMmotorstarter[1].et200SpMotorstarterInputs[0..1].iActBit1 := FALSE;
   Et200SpMotorstarterInterfaceAllUnits[0].EMmotorstarter[2].et200SpMotorstarterInputs[0..1].iActBit1 := FALSE;
   Et200SpMotorstarterInterfaceAllUnits[0].EMmotorstarter[3].et200SpMotorstarterInputs[0..1].iActBit1 := FALSE;
   Et200SpMotorstarterInterfaceAllUnits[0].EMmotorstarter[4].et200SpMotorstarterInputs[0..1].iActBit1 := FALSE;
   Et200SpMotorstarterInterfaceAllUnits[0].EMmotorstarter[5].et200SpMotorstarterInputs[0..1].iActBit1 := FALSE;
   Et200SpMotorstarterInterfaceAllUnits[0].EMmotorstarter[6].et200SpMotorstarterInputs[0..1].iActBit1 := FALSE;
   Et200SpMotorstarterInterfaceAllUnits[0].EMmotorstarter[7].et200SpMotorstarterInputs[0..1].iActBit1 := FALSE;
   Et200SpMotorstarterInterfaceAllUnits[0].EMmotorstarter[0].et200SpMotorstarterInputs[0..1].iActBit2 := FALSE;
   Et200SpMotorstarterInterfaceAllUnits[0].EMmotorstarter[1].et200SpMotorstarterInputs[0..1].iActBit2 := FALSE;
   Et200SpMotorstarterInterfaceAllUnits[0].EMmotorstarter[2].et200SpMotorstarterInputs[0..1].iActBit2 := FALSE;
   Et200SpMotorstarterInterfaceAllUnits[0].EMmotorstarter[3].et200SpMotorstarterInputs[0..1].iActBit2 := FALSE;
   Et200SpMotorstarterInterfaceAllUnits[0].EMmotorstarter[4].et200SpMotorstarterInputs[0..1].iActBit2 := FALSE;
   Et200SpMotorstarterInterfaceAllUnits[0].EMmotorstarter[5].et200SpMotorstarterInputs[0..1].iActBit2 := FALSE;
   Et200SpMotorstarterInterfaceAllUnits[0].EMmotorstarter[6].et200SpMotorstarterInputs[0..1].iActBit2 := FALSE;
   Et200SpMotorstarterInterfaceAllUnits[0].EMmotorstarter[7].et200SpMotorstarterInputs[0..1].iActBit2 := FALSE;
   Et200SpMotorstarterInterfaceAllUnits[0].EMmotorstarter[0].et200SpMotorstarterInputs[0..1].iActBit3 := FALSE;
   Et200SpMotorstarterInterfaceAllUnits[0].EMmotorstarter[1].et200SpMotorstarterInputs[0..1].iActBit3 := FALSE;
   Et200SpMotorstarterInterfaceAllUnits[0].EMmotorstarter[2].et200SpMotorstarterInputs[0..1].iActBit3 := FALSE;
   Et200SpMotorstarterInterfaceAllUnits[0].EMmotorstarter[3].et200SpMotorstarterInputs[0..1].iActBit3 := FALSE;
   Et200SpMotorstarterInterfaceAllUnits[0].EMmotorstarter[4].et200SpMotorstarterInputs[0..1].iActBit3 := FALSE;
   Et200SpMotorstarterInterfaceAllUnits[0].EMmotorstarter[5].et200SpMotorstarterInputs[0..1].iActBit3 := FALSE;
   Et200SpMotorstarterInterfaceAllUnits[0].EMmotorstarter[6].et200SpMotorstarterInputs[0..1].iActBit3 := FALSE;
   Et200SpMotorstarterInterfaceAllUnits[0].EMmotorstarter[7].et200SpMotorstarterInputs[0..1].iActBit3 := FALSE;
   Et200SpMotorstarterInterfaceAllUnits[0].EMmotorstarter[0].et200SpMotorstarterInputs[0..1].iActBit4 := FALSE;
   Et200SpMotorstarterInterfaceAllUnits[0].EMmotorstarter[1].et200SpMotorstarterInputs[0..1].iActBit4 := FALSE;
   Et200SpMotorstarterInterfaceAllUnits[0].EMmotorstarter[2].et200SpMotorstarterInputs[0..1].iActBit4 := FALSE;
   Et200SpMotorstarterInterfaceAllUnits[0].EMmotorstarter[3].et200SpMotorstarterInputs[0..1].iActBit4 := FALSE;
   Et200SpMotorstarterInterfaceAllUnits[0].EMmotorstarter[4].et200SpMotorstarterInputs[0..1].iActBit4 := FALSE;
   Et200SpMotorstarterInterfaceAllUnits[0].EMmotorstarter[5].et200SpMotorstarterInputs[0..1].iActBit4 := FALSE;
   Et200SpMotorstarterInterfaceAllUnits[0].EMmotorstarter[6].et200SpMotorstarterInputs[0..1].iActBit4 := FALSE;
   Et200SpMotorstarterInterfaceAllUnits[0].EMmotorstarter[7].et200SpMotorstarterInputs[0..1].iActBit4 := FALSE;
   Et200SpMotorstarterInterfaceAllUnits[0].EMmotorstarter[0].et200SpMotorstarterInputs[0..1].iActBit5 := FALSE;
   Et200SpMotorstarterInterfaceAllUnits[0].EMmotorstarter[1].et200SpMotorstarterInputs[0..1].iActBit5 := FALSE;
   Et200SpMotorstarterInterfaceAllUnits[0].EMmotorstarter[2].et200SpMotorstarterInputs[0..1].iActBit5 := FALSE;
   Et200SpMotorstarterInterfaceAllUnits[0].EMmotorstarter[3].et200SpMotorstarterInputs[0..1].iActBit5 := FALSE;
   Et200SpMotorstarterInterfaceAllUnits[0].EMmotorstarter[4].et200SpMotorstarterInputs[0..1].iActBit5 := FALSE;
   Et200SpMotorstarterInterfaceAllUnits[0].EMmotorstarter[5].et200SpMotorstarterInputs[0..1].iActBit5 := FALSE;
   Et200SpMotorstarterInterfaceAllUnits[0].EMmotorstarter[6].et200SpMotorstarterInputs[0..1].iActBit5 := FALSE;
   Et200SpMotorstarterInterfaceAllUnits[0].EMmotorstarter[7].et200SpMotorstarterInputs[0..1].iActBit5 := FALSE;
   Et200SpMotorstarterInterfaceAllUnits[0].EMmotorstarter[0].et200SpMotorstarterInputs[0..1].manualOperating := FALSE;
   Et200SpMotorstarterInterfaceAllUnits[0].EMmotorstarter[1].et200SpMotorstarterInputs[0..1].manualOperating := FALSE;
   Et200SpMotorstarterInterfaceAllUnits[0].EMmotorstarter[2].et200SpMotorstarterInputs[0..1].manualOperating := FALSE;
   Et200SpMotorstarterInterfaceAllUnits[0].EMmotorstarter[3].et200SpMotorstarterInputs[0..1].manualOperating := FALSE;
   Et200SpMotorstarterInterfaceAllUnits[0].EMmotorstarter[4].et200SpMotorstarterInputs[0..1].manualOperating := FALSE;
   Et200SpMotorstarterInterfaceAllUnits[0].EMmotorstarter[5].et200SpMotorstarterInputs[0..1].manualOperating := FALSE;
   Et200SpMotorstarterInterfaceAllUnits[0].EMmotorstarter[6].et200SpMotorstarterInputs[0..1].manualOperating := FALSE;
   Et200SpMotorstarterInterfaceAllUnits[0].EMmotorstarter[7].et200SpMotorstarterInputs[0..1].manualOperating := FALSE;
   Et200SpMotorstarterInterfaceAllUnits[0].EMmotorstarter[0].et200SpMotorstarterInputs[0..1].spare1 := FALSE;
   Et200SpMotorstarterInterfaceAllUnits[0].EMmotorstarter[1].et200SpMotorstarterInputs[0..1].spare1 := FALSE;
   Et200SpMotorstarterInterfaceAllUnits[0].EMmotorstarter[2].et200SpMotorstarterInputs[0..1].spare1 := FALSE;
   Et200SpMotorstarterInterfaceAllUnits[0].EMmotorstarter[3].et200SpMotorstarterInputs[0..1].spare1 := FALSE;
   Et200SpMotorstarterInterfaceAllUnits[0].EMmotorstarter[4].et200SpMotorstarterInputs[0..1].spare1 := FALSE;
   Et200SpMotorstarterInterfaceAllUnits[0].EMmotorstarter[5].et200SpMotorstarterInputs[0..1].spare1 := FALSE;
   Et200SpMotorstarterInterfaceAllUnits[0].EMmotorstarter[6].et200SpMotorstarterInputs[0..1].spare1 := FALSE;
   Et200SpMotorstarterInterfaceAllUnits[0].EMmotorstarter[7].et200SpMotorstarterInputs[0..1].spare1 := FALSE;
   Et200SpMotorstarterInterfaceAllUnits[0].EMmotorstarter[0].et200SpMotorstarterInputs[0..1].readyStartOn := FALSE;
   Et200SpMotorstarterInterfaceAllUnits[0].EMmotorstarter[1].et200SpMotorstarterInputs[0..1].readyStartOn := FALSE;
   Et200SpMotorstarterInterfaceAllUnits[0].EMmotorstarter[2].et200SpMotorstarterInputs[0..1].readyStartOn := FALSE;
   Et200SpMotorstarterInterfaceAllUnits[0].EMmotorstarter[3].et200SpMotorstarterInputs[0..1].readyStartOn := FALSE;
   Et200SpMotorstarterInterfaceAllUnits[0].EMmotorstarter[4].et200SpMotorstarterInputs[0..1].readyStartOn := FALSE;
   Et200SpMotorstarterInterfaceAllUnits[0].EMmotorstarter[5].et200SpMotorstarterInputs[0..1].readyStartOn := FALSE;
   Et200SpMotorstarterInterfaceAllUnits[0].EMmotorstarter[6].et200SpMotorstarterInputs[0..1].readyStartOn := FALSE;
   Et200SpMotorstarterInterfaceAllUnits[0].EMmotorstarter[7].et200SpMotorstarterInputs[0..1].readyStartOn := FALSE;
   Et200SpMotorstarterInterfaceAllUnits[0].EMmotorstarter[0].et200SpMotorstarterInputs[0..1].motorOnRight := FALSE;
   Et200SpMotorstarterInterfaceAllUnits[0].EMmotorstarter[1].et200SpMotorstarterInputs[0..1].motorOnRight := FALSE;
   Et200SpMotorstarterInterfaceAllUnits[0].EMmotorstarter[2].et200SpMotorstarterInputs[0..1].motorOnRight := FALSE;
   Et200SpMotorstarterInterfaceAllUnits[0].EMmotorstarter[3].et200SpMotorstarterInputs[0..1].motorOnRight := FALSE;
   Et200SpMotorstarterInterfaceAllUnits[0].EMmotorstarter[4].et200SpMotorstarterInputs[0..1].motorOnRight := FALSE;
   Et200SpMotorstarterInterfaceAllUnits[0].EMmotorstarter[5].et200SpMotorstarterInputs[0..1].motorOnRight := FALSE;
   Et200SpMotorstarterInterfaceAllUnits[0].EMmotorstarter[6].et200SpMotorstarterInputs[0..1].motorOnRight := FALSE;
   Et200SpMotorstarterInterfaceAllUnits[0].EMmotorstarter[7].et200SpMotorstarterInputs[0..1].motorOnRight := FALSE;
   Et200SpMotorstarterInterfaceAllUnits[0].EMmotorstarter[0].et200SpMotorstarterInputs[0..1].motorOnLeft := FALSE;
   Et200SpMotorstarterInterfaceAllUnits[0].EMmotorstarter[1].et200SpMotorstarterInputs[0..1].motorOnLeft := FALSE;
   Et200SpMotorstarterInterfaceAllUnits[0].EMmotorstarter[2].et200SpMotorstarterInputs[0..1].motorOnLeft := FALSE;
   Et200SpMotorstarterInterfaceAllUnits[0].EMmotorstarter[3].et200SpMotorstarterInputs[0..1].motorOnLeft := FALSE;
   Et200SpMotorstarterInterfaceAllUnits[0].EMmotorstarter[4].et200SpMotorstarterInputs[0..1].motorOnLeft := FALSE;
   Et200SpMotorstarterInterfaceAllUnits[0].EMmotorstarter[5].et200SpMotorstarterInputs[0..1].motorOnLeft := FALSE;
   Et200SpMotorstarterInterfaceAllUnits[0].EMmotorstarter[6].et200SpMotorstarterInputs[0..1].motorOnLeft := FALSE;
   Et200SpMotorstarterInterfaceAllUnits[0].EMmotorstarter[7].et200SpMotorstarterInputs[0..1].motorOnLeft := FALSE;
   Et200SpMotorstarterInterfaceAllUnits[0].EMmotorstarter[0].et200SpMotorstarterInputs[0..1].quickstopActive := FALSE;
   Et200SpMotorstarterInterfaceAllUnits[0].EMmotorstarter[1].et200SpMotorstarterInputs[0..1].quickstopActive := FALSE;
   Et200SpMotorstarterInterfaceAllUnits[0].EMmotorstarter[2].et200SpMotorstarterInputs[0..1].quickstopActive := FALSE;
   Et200SpMotorstarterInterfaceAllUnits[0].EMmotorstarter[3].et200SpMotorstarterInputs[0..1].quickstopActive := FALSE;
   Et200SpMotorstarterInterfaceAllUnits[0].EMmotorstarter[4].et200SpMotorstarterInputs[0..1].quickstopActive := FALSE;
   Et200SpMotorstarterInterfaceAllUnits[0].EMmotorstarter[5].et200SpMotorstarterInputs[0..1].quickstopActive := FALSE;
   Et200SpMotorstarterInterfaceAllUnits[0].EMmotorstarter[6].et200SpMotorstarterInputs[0..1].quickstopActive := FALSE;
   Et200SpMotorstarterInterfaceAllUnits[0].EMmotorstarter[7].et200SpMotorstarterInputs[0..1].quickstopActive := FALSE;
   Et200SpMotorstarterInterfaceAllUnits[0].EMmotorstarter[0].et200SpMotorstarterInputs[0..1].energySaving := FALSE;
   Et200SpMotorstarterInterfaceAllUnits[0].EMmotorstarter[1].et200SpMotorstarterInputs[0..1].energySaving := FALSE;
   Et200SpMotorstarterInterfaceAllUnits[0].EMmotorstarter[2].et200SpMotorstarterInputs[0..1].energySaving := FALSE;
   Et200SpMotorstarterInterfaceAllUnits[0].EMmotorstarter[3].et200SpMotorstarterInputs[0..1].energySaving := FALSE;
   Et200SpMotorstarterInterfaceAllUnits[0].EMmotorstarter[4].et200SpMotorstarterInputs[0..1].energySaving := FALSE;
   Et200SpMotorstarterInterfaceAllUnits[0].EMmotorstarter[5].et200SpMotorstarterInputs[0..1].energySaving := FALSE;
   Et200SpMotorstarterInterfaceAllUnits[0].EMmotorstarter[6].et200SpMotorstarterInputs[0..1].energySaving := FALSE;
   Et200SpMotorstarterInterfaceAllUnits[0].EMmotorstarter[7].et200SpMotorstarterInputs[0..1].energySaving := FALSE;
   Et200SpMotorstarterInterfaceAllUnits[0].EMmotorstarter[0].et200SpMotorstarterInputs[0..1].moduleInserted := FALSE;
   Et200SpMotorstarterInterfaceAllUnits[0].EMmotorstarter[1].et200SpMotorstarterInputs[0..1].moduleInserted := FALSE;
   Et200SpMotorstarterInterfaceAllUnits[0].EMmotorstarter[2].et200SpMotorstarterInputs[0..1].moduleInserted := FALSE;
   Et200SpMotorstarterInterfaceAllUnits[0].EMmotorstarter[3].et200SpMotorstarterInputs[0..1].moduleInserted := FALSE;
   Et200SpMotorstarterInterfaceAllUnits[0].EMmotorstarter[4].et200SpMotorstarterInputs[0..1].moduleInserted := FALSE;
   Et200SpMotorstarterInterfaceAllUnits[0].EMmotorstarter[5].et200SpMotorstarterInputs[0..1].moduleInserted := FALSE;
   Et200SpMotorstarterInterfaceAllUnits[0].EMmotorstarter[6].et200SpMotorstarterInputs[0..1].moduleInserted := FALSE;
   Et200SpMotorstarterInterfaceAllUnits[0].EMmotorstarter[7].et200SpMotorstarterInputs[0..1].moduleInserted := FALSE;
   Et200SpMotorstarterInterfaceAllUnits[0].EMmotorstarter[0].et200SpMotorstarterInputs[0..1].exProtectionMotorActive := FALSE;
   Et200SpMotorstarterInterfaceAllUnits[0].EMmotorstarter[1].et200SpMotorstarterInputs[0..1].exProtectionMotorActive := FALSE;
   Et200SpMotorstarterInterfaceAllUnits[0].EMmotorstarter[2].et200SpMotorstarterInputs[0..1].exProtectionMotorActive := FALSE;
   Et200SpMotorstarterInterfaceAllUnits[0].EMmotorstarter[3].et200SpMotorstarterInputs[0..1].exProtectionMotorActive := FALSE;
   Et200SpMotorstarterInterfaceAllUnits[0].EMmotorstarter[4].et200SpMotorstarterInputs[0..1].exProtectionMotorActive := FALSE;
   Et200SpMotorstarterInterfaceAllUnits[0].EMmotorstarter[5].et200SpMotorstarterInputs[0..1].exProtectionMotorActive := FALSE;
   Et200SpMotorstarterInterfaceAllUnits[0].EMmotorstarter[6].et200SpMotorstarterInputs[0..1].exProtectionMotorActive := FALSE;
   Et200SpMotorstarterInterfaceAllUnits[0].EMmotorstarter[7].et200SpMotorstarterInputs[0..1].exProtectionMotorActive := FALSE;
   Et200SpMotorstarterInterfaceAllUnits[0].EMmotorstarter[0].et200SpMotorstarterInputs[0..1].blockActive := FALSE;
   Et200SpMotorstarterInterfaceAllUnits[0].EMmotorstarter[1].et200SpMotorstarterInputs[0..1].blockActive := FALSE;
   Et200SpMotorstarterInterfaceAllUnits[0].EMmotorstarter[2].et200SpMotorstarterInputs[0..1].blockActive := FALSE;
   Et200SpMotorstarterInterfaceAllUnits[0].EMmotorstarter[3].et200SpMotorstarterInputs[0..1].blockActive := FALSE;
   Et200SpMotorstarterInterfaceAllUnits[0].EMmotorstarter[4].et200SpMotorstarterInputs[0..1].blockActive := FALSE;
   Et200SpMotorstarterInterfaceAllUnits[0].EMmotorstarter[5].et200SpMotorstarterInputs[0..1].blockActive := FALSE;
   Et200SpMotorstarterInterfaceAllUnits[0].EMmotorstarter[6].et200SpMotorstarterInputs[0..1].blockActive := FALSE;
   Et200SpMotorstarterInterfaceAllUnits[0].EMmotorstarter[7].et200SpMotorstarterInputs[0..1].blockActive := FALSE;
   Et200SpMotorstarterInterfaceAllUnits[0].EMmotorstarter[0].et200SpMotorstarterInputs[0..1].thermalMotorOverload := FALSE;
   Et200SpMotorstarterInterfaceAllUnits[0].EMmotorstarter[1].et200SpMotorstarterInputs[0..1].thermalMotorOverload := FALSE;
   Et200SpMotorstarterInterfaceAllUnits[0].EMmotorstarter[2].et200SpMotorstarterInputs[0..1].thermalMotorOverload := FALSE;
   Et200SpMotorstarterInterfaceAllUnits[0].EMmotorstarter[3].et200SpMotorstarterInputs[0..1].thermalMotorOverload := FALSE;
   Et200SpMotorstarterInterfaceAllUnits[0].EMmotorstarter[4].et200SpMotorstarterInputs[0..1].thermalMotorOverload := FALSE;
   Et200SpMotorstarterInterfaceAllUnits[0].EMmotorstarter[5].et200SpMotorstarterInputs[0..1].thermalMotorOverload := FALSE;
   Et200SpMotorstarterInterfaceAllUnits[0].EMmotorstarter[6].et200SpMotorstarterInputs[0..1].thermalMotorOverload := FALSE;
   Et200SpMotorstarterInterfaceAllUnits[0].EMmotorstarter[7].et200SpMotorstarterInputs[0..1].thermalMotorOverload := FALSE;
   Et200SpMotorstarterInterfaceAllUnits[0].EMmotorstarter[0].et200SpMotorstarterInputs[0..1].spare5 := FALSE;
   Et200SpMotorstarterInterfaceAllUnits[0].EMmotorstarter[1].et200SpMotorstarterInputs[0..1].spare5 := FALSE;
   Et200SpMotorstarterInterfaceAllUnits[0].EMmotorstarter[2].et200SpMotorstarterInputs[0..1].spare5 := FALSE;
   Et200SpMotorstarterInterfaceAllUnits[0].EMmotorstarter[3].et200SpMotorstarterInputs[0..1].spare5 := FALSE;
   Et200SpMotorstarterInterfaceAllUnits[0].EMmotorstarter[4].et200SpMotorstarterInputs[0..1].spare5 := FALSE;
   Et200SpMotorstarterInterfaceAllUnits[0].EMmotorstarter[5].et200SpMotorstarterInputs[0..1].spare5 := FALSE;
   Et200SpMotorstarterInterfaceAllUnits[0].EMmotorstarter[6].et200SpMotorstarterInputs[0..1].spare5 := FALSE;
   Et200SpMotorstarterInterfaceAllUnits[0].EMmotorstarter[7].et200SpMotorstarterInputs[0..1].spare5 := FALSE;
   Et200SpMotorstarterInterfaceAllUnits[0].EMmotorstarter[0].et200SpMotorstarterInputs[0..1].currentLimitTripping := FALSE;
   Et200SpMotorstarterInterfaceAllUnits[0].EMmotorstarter[1].et200SpMotorstarterInputs[0..1].currentLimitTripping := FALSE;
   Et200SpMotorstarterInterfaceAllUnits[0].EMmotorstarter[2].et200SpMotorstarterInputs[0..1].currentLimitTripping := FALSE;
   Et200SpMotorstarterInterfaceAllUnits[0].EMmotorstarter[3].et200SpMotorstarterInputs[0..1].currentLimitTripping := FALSE;
   Et200SpMotorstarterInterfaceAllUnits[0].EMmotorstarter[4].et200SpMotorstarterInputs[0..1].currentLimitTripping := FALSE;
   Et200SpMotorstarterInterfaceAllUnits[0].EMmotorstarter[5].et200SpMotorstarterInputs[0..1].currentLimitTripping := FALSE;
   Et200SpMotorstarterInterfaceAllUnits[0].EMmotorstarter[6].et200SpMotorstarterInputs[0..1].currentLimitTripping := FALSE;
   Et200SpMotorstarterInterfaceAllUnits[0].EMmotorstarter[7].et200SpMotorstarterInputs[0..1].currentLimitTripping := FALSE;
   Et200SpMotorstarterInterfaceAllUnits[0].EMmotorstarter[0].et200SpMotorstarterInputs[0..1].statusFailDi := FALSE;
   Et200SpMotorstarterInterfaceAllUnits[0].EMmotorstarter[1].et200SpMotorstarterInputs[0..1].statusFailDi := FALSE;
   Et200SpMotorstarterInterfaceAllUnits[0].EMmotorstarter[2].et200SpMotorstarterInputs[0..1].statusFailDi := FALSE;
   Et200SpMotorstarterInterfaceAllUnits[0].EMmotorstarter[3].et200SpMotorstarterInputs[0..1].statusFailDi := FALSE;
   Et200SpMotorstarterInterfaceAllUnits[0].EMmotorstarter[4].et200SpMotorstarterInputs[0..1].statusFailDi := FALSE;
   Et200SpMotorstarterInterfaceAllUnits[0].EMmotorstarter[5].et200SpMotorstarterInputs[0..1].statusFailDi := FALSE;
   Et200SpMotorstarterInterfaceAllUnits[0].EMmotorstarter[6].et200SpMotorstarterInputs[0..1].statusFailDi := FALSE;
   Et200SpMotorstarterInterfaceAllUnits[0].EMmotorstarter[7].et200SpMotorstarterInputs[0..1].statusFailDi := FALSE;
   Et200SpMotorstarterInterfaceAllUnits[0].EMmotorstarter[0].et200SpMotorstarterInputs[0..1].residualCurrent := FALSE;
   Et200SpMotorstarterInterfaceAllUnits[0].EMmotorstarter[1].et200SpMotorstarterInputs[0..1].residualCurrent := FALSE;
   Et200SpMotorstarterInterfaceAllUnits[0].EMmotorstarter[2].et200SpMotorstarterInputs[0..1].residualCurrent := FALSE;
   Et200SpMotorstarterInterfaceAllUnits[0].EMmotorstarter[3].et200SpMotorstarterInputs[0..1].residualCurrent := FALSE;
   Et200SpMotorstarterInterfaceAllUnits[0].EMmotorstarter[4].et200SpMotorstarterInputs[0..1].residualCurrent := FALSE;
   Et200SpMotorstarterInterfaceAllUnits[0].EMmotorstarter[5].et200SpMotorstarterInputs[0..1].residualCurrent := FALSE;
   Et200SpMotorstarterInterfaceAllUnits[0].EMmotorstarter[6].et200SpMotorstarterInputs[0..1].residualCurrent := FALSE;
   Et200SpMotorstarterInterfaceAllUnits[0].EMmotorstarter[7].et200SpMotorstarterInputs[0..1].residualCurrent := FALSE;
   Et200SpMotorstarterInterfaceAllUnits[0].EMmotorstarter[0].et200SpMotorstarterInputs[0..1].asymmetryDetected := FALSE;
   Et200SpMotorstarterInterfaceAllUnits[0].EMmotorstarter[1].et200SpMotorstarterInputs[0..1].asymmetryDetected := FALSE;
   Et200SpMotorstarterInterfaceAllUnits[0].EMmotorstarter[2].et200SpMotorstarterInputs[0..1].asymmetryDetected := FALSE;
   Et200SpMotorstarterInterfaceAllUnits[0].EMmotorstarter[3].et200SpMotorstarterInputs[0..1].asymmetryDetected := FALSE;
   Et200SpMotorstarterInterfaceAllUnits[0].EMmotorstarter[4].et200SpMotorstarterInputs[0..1].asymmetryDetected := FALSE;
   Et200SpMotorstarterInterfaceAllUnits[0].EMmotorstarter[5].et200SpMotorstarterInputs[0..1].asymmetryDetected := FALSE;
   Et200SpMotorstarterInterfaceAllUnits[0].EMmotorstarter[6].et200SpMotorstarterInputs[0..1].asymmetryDetected := FALSE;
   Et200SpMotorstarterInterfaceAllUnits[0].EMmotorstarter[7].et200SpMotorstarterInputs[0..1].asymmetryDetected := FALSE;
   Et200SpMotorstarterInterfaceAllUnits[0].EMmotorstarter[0].et200SpMotorstarterInputs[0..1].overtemperature := FALSE;
   Et200SpMotorstarterInterfaceAllUnits[0].EMmotorstarter[1].et200SpMotorstarterInputs[0..1].overtemperature := FALSE;
   Et200SpMotorstarterInterfaceAllUnits[0].EMmotorstarter[2].et200SpMotorstarterInputs[0..1].overtemperature := FALSE;
   Et200SpMotorstarterInterfaceAllUnits[0].EMmotorstarter[3].et200SpMotorstarterInputs[0..1].overtemperature := FALSE;
   Et200SpMotorstarterInterfaceAllUnits[0].EMmotorstarter[4].et200SpMotorstarterInputs[0..1].overtemperature := FALSE;
   Et200SpMotorstarterInterfaceAllUnits[0].EMmotorstarter[5].et200SpMotorstarterInputs[0..1].overtemperature := FALSE;
   Et200SpMotorstarterInterfaceAllUnits[0].EMmotorstarter[6].et200SpMotorstarterInputs[0..1].overtemperature := FALSE;
   Et200SpMotorstarterInterfaceAllUnits[0].EMmotorstarter[7].et200SpMotorstarterInputs[0..1].overtemperature := FALSE;
   Et200SpMotorstarterInterfaceAllUnits[0].EMmotorstarter[0].et200SpMotorstarterInputs[0..1].spare7 := FALSE;
   Et200SpMotorstarterInterfaceAllUnits[0].EMmotorstarter[1].et200SpMotorstarterInputs[0..1].spare7 := FALSE;
   Et200SpMotorstarterInterfaceAllUnits[0].EMmotorstarter[2].et200SpMotorstarterInputs[0..1].spare7 := FALSE;
   Et200SpMotorstarterInterfaceAllUnits[0].EMmotorstarter[3].et200SpMotorstarterInputs[0..1].spare7 := FALSE;
   Et200SpMotorstarterInterfaceAllUnits[0].EMmotorstarter[4].et200SpMotorstarterInputs[0..1].spare7 := FALSE;
   Et200SpMotorstarterInterfaceAllUnits[0].EMmotorstarter[5].et200SpMotorstarterInputs[0..1].spare7 := FALSE;
   Et200SpMotorstarterInterfaceAllUnits[0].EMmotorstarter[6].et200SpMotorstarterInputs[0..1].spare7 := FALSE;
   Et200SpMotorstarterInterfaceAllUnits[0].EMmotorstarter[7].et200SpMotorstarterInputs[0..1].spare7 := FALSE;
   Et200SpMotorstarterInterfaceAllUnits[0].EMmotorstarter[0].et200SpMotorstarterOutputs[0..1].motorCw := FALSE;
   Et200SpMotorstarterInterfaceAllUnits[0].EMmotorstarter[1].et200SpMotorstarterOutputs[0..1].motorCw := FALSE;
   Et200SpMotorstarterInterfaceAllUnits[0].EMmotorstarter[2].et200SpMotorstarterOutputs[0..1].motorCw := FALSE;
   Et200SpMotorstarterInterfaceAllUnits[0].EMmotorstarter[3].et200SpMotorstarterOutputs[0..1].motorCw := FALSE;
   Et200SpMotorstarterInterfaceAllUnits[0].EMmotorstarter[4].et200SpMotorstarterOutputs[0..1].motorCw := FALSE;
   Et200SpMotorstarterInterfaceAllUnits[0].EMmotorstarter[5].et200SpMotorstarterOutputs[0..1].motorCw := FALSE;
   Et200SpMotorstarterInterfaceAllUnits[0].EMmotorstarter[6].et200SpMotorstarterOutputs[0..1].motorCw := FALSE;
   Et200SpMotorstarterInterfaceAllUnits[0].EMmotorstarter[7].et200SpMotorstarterOutputs[0..1].motorCw := FALSE;
   Et200SpMotorstarterInterfaceAllUnits[0].EMmotorstarter[0].et200SpMotorstarterOutputs[0..1].motorCww := FALSE;
   Et200SpMotorstarterInterfaceAllUnits[0].EMmotorstarter[1].et200SpMotorstarterOutputs[0..1].motorCww := FALSE;
   Et200SpMotorstarterInterfaceAllUnits[0].EMmotorstarter[2].et200SpMotorstarterOutputs[0..1].motorCww := FALSE;
   Et200SpMotorstarterInterfaceAllUnits[0].EMmotorstarter[3].et200SpMotorstarterOutputs[0..1].motorCww := FALSE;
   Et200SpMotorstarterInterfaceAllUnits[0].EMmotorstarter[4].et200SpMotorstarterOutputs[0..1].motorCww := FALSE;
   Et200SpMotorstarterInterfaceAllUnits[0].EMmotorstarter[5].et200SpMotorstarterOutputs[0..1].motorCww := FALSE;
   Et200SpMotorstarterInterfaceAllUnits[0].EMmotorstarter[6].et200SpMotorstarterOutputs[0..1].motorCww := FALSE;
   Et200SpMotorstarterInterfaceAllUnits[0].EMmotorstarter[7].et200SpMotorstarterOutputs[0..1].motorCww := FALSE;
   Et200SpMotorstarterInterfaceAllUnits[0].EMmotorstarter[0].et200SpMotorstarterOutputs[0..1].reserve1 := FALSE;
   Et200SpMotorstarterInterfaceAllUnits[0].EMmotorstarter[1].et200SpMotorstarterOutputs[0..1].reserve1 := FALSE;
   Et200SpMotorstarterInterfaceAllUnits[0].EMmotorstarter[2].et200SpMotorstarterOutputs[0..1].reserve1 := FALSE;
   Et200SpMotorstarterInterfaceAllUnits[0].EMmotorstarter[3].et200SpMotorstarterOutputs[0..1].reserve1 := FALSE;
   Et200SpMotorstarterInterfaceAllUnits[0].EMmotorstarter[4].et200SpMotorstarterOutputs[0..1].reserve1 := FALSE;
   Et200SpMotorstarterInterfaceAllUnits[0].EMmotorstarter[5].et200SpMotorstarterOutputs[0..1].reserve1 := FALSE;
   Et200SpMotorstarterInterfaceAllUnits[0].EMmotorstarter[6].et200SpMotorstarterOutputs[0..1].reserve1 := FALSE;
   Et200SpMotorstarterInterfaceAllUnits[0].EMmotorstarter[7].et200SpMotorstarterOutputs[0..1].reserve1 := FALSE;
   Et200SpMotorstarterInterfaceAllUnits[0].EMmotorstarter[0].et200SpMotorstarterOutputs[0..1].tripReset := FALSE;
   Et200SpMotorstarterInterfaceAllUnits[0].EMmotorstarter[1].et200SpMotorstarterOutputs[0..1].tripReset := FALSE;
   Et200SpMotorstarterInterfaceAllUnits[0].EMmotorstarter[2].et200SpMotorstarterOutputs[0..1].tripReset := FALSE;
   Et200SpMotorstarterInterfaceAllUnits[0].EMmotorstarter[3].et200SpMotorstarterOutputs[0..1].tripReset := FALSE;
   Et200SpMotorstarterInterfaceAllUnits[0].EMmotorstarter[4].et200SpMotorstarterOutputs[0..1].tripReset := FALSE;
   Et200SpMotorstarterInterfaceAllUnits[0].EMmotorstarter[5].et200SpMotorstarterOutputs[0..1].tripReset := FALSE;
   Et200SpMotorstarterInterfaceAllUnits[0].EMmotorstarter[6].et200SpMotorstarterOutputs[0..1].tripReset := FALSE;
   Et200SpMotorstarterInterfaceAllUnits[0].EMmotorstarter[7].et200SpMotorstarterOutputs[0..1].tripReset := FALSE;
   Et200SpMotorstarterInterfaceAllUnits[0].EMmotorstarter[0].et200SpMotorstarterOutputs[0..1].emergencyStart := FALSE;
   Et200SpMotorstarterInterfaceAllUnits[0].EMmotorstarter[1].et200SpMotorstarterOutputs[0..1].emergencyStart := FALSE;
   Et200SpMotorstarterInterfaceAllUnits[0].EMmotorstarter[2].et200SpMotorstarterOutputs[0..1].emergencyStart := FALSE;
   Et200SpMotorstarterInterfaceAllUnits[0].EMmotorstarter[3].et200SpMotorstarterOutputs[0..1].emergencyStart := FALSE;
   Et200SpMotorstarterInterfaceAllUnits[0].EMmotorstarter[4].et200SpMotorstarterOutputs[0..1].emergencyStart := FALSE;
   Et200SpMotorstarterInterfaceAllUnits[0].EMmotorstarter[5].et200SpMotorstarterOutputs[0..1].emergencyStart := FALSE;
   Et200SpMotorstarterInterfaceAllUnits[0].EMmotorstarter[6].et200SpMotorstarterOutputs[0..1].emergencyStart := FALSE;
   Et200SpMotorstarterInterfaceAllUnits[0].EMmotorstarter[7].et200SpMotorstarterOutputs[0..1].emergencyStart := FALSE;
   Et200SpMotorstarterInterfaceAllUnits[0].EMmotorstarter[0].et200SpMotorstarterOutputs[0..1].reserve2 := FALSE;
   Et200SpMotorstarterInterfaceAllUnits[0].EMmotorstarter[1].et200SpMotorstarterOutputs[0..1].reserve2 := FALSE;
   Et200SpMotorstarterInterfaceAllUnits[0].EMmotorstarter[2].et200SpMotorstarterOutputs[0..1].reserve2 := FALSE;
   Et200SpMotorstarterInterfaceAllUnits[0].EMmotorstarter[3].et200SpMotorstarterOutputs[0..1].reserve2 := FALSE;
   Et200SpMotorstarterInterfaceAllUnits[0].EMmotorstarter[4].et200SpMotorstarterOutputs[0..1].reserve2 := FALSE;
   Et200SpMotorstarterInterfaceAllUnits[0].EMmotorstarter[5].et200SpMotorstarterOutputs[0..1].reserve2 := FALSE;
   Et200SpMotorstarterInterfaceAllUnits[0].EMmotorstarter[6].et200SpMotorstarterOutputs[0..1].reserve2 := FALSE;
   Et200SpMotorstarterInterfaceAllUnits[0].EMmotorstarter[7].et200SpMotorstarterOutputs[0..1].reserve2 := FALSE;
   Et200SpMotorstarterInterfaceAllUnits[0].EMmotorstarter[0].et200SpMotorstarterOutputs[0..1].reserve3 := FALSE;
   Et200SpMotorstarterInterfaceAllUnits[0].EMmotorstarter[1].et200SpMotorstarterOutputs[0..1].reserve3 := FALSE;
   Et200SpMotorstarterInterfaceAllUnits[0].EMmotorstarter[2].et200SpMotorstarterOutputs[0..1].reserve3 := FALSE;
   Et200SpMotorstarterInterfaceAllUnits[0].EMmotorstarter[3].et200SpMotorstarterOutputs[0..1].reserve3 := FALSE;
   Et200SpMotorstarterInterfaceAllUnits[0].EMmotorstarter[4].et200SpMotorstarterOutputs[0..1].reserve3 := FALSE;
   Et200SpMotorstarterInterfaceAllUnits[0].EMmotorstarter[5].et200SpMotorstarterOutputs[0..1].reserve3 := FALSE;
   Et200SpMotorstarterInterfaceAllUnits[0].EMmotorstarter[6].et200SpMotorstarterOutputs[0..1].reserve3 := FALSE;
   Et200SpMotorstarterInterfaceAllUnits[0].EMmotorstarter[7].et200SpMotorstarterOutputs[0..1].reserve3 := FALSE;
   Et200SpMotorstarterInterfaceAllUnits[0].EMmotorstarter[0].et200SpMotorstarterOutputs[0..1].coldStart := FALSE;
   Et200SpMotorstarterInterfaceAllUnits[0].EMmotorstarter[1].et200SpMotorstarterOutputs[0..1].coldStart := FALSE;
   Et200SpMotorstarterInterfaceAllUnits[0].EMmotorstarter[2].et200SpMotorstarterOutputs[0..1].coldStart := FALSE;
   Et200SpMotorstarterInterfaceAllUnits[0].EMmotorstarter[3].et200SpMotorstarterOutputs[0..1].coldStart := FALSE;
   Et200SpMotorstarterInterfaceAllUnits[0].EMmotorstarter[4].et200SpMotorstarterOutputs[0..1].coldStart := FALSE;
   Et200SpMotorstarterInterfaceAllUnits[0].EMmotorstarter[5].et200SpMotorstarterOutputs[0..1].coldStart := FALSE;
   Et200SpMotorstarterInterfaceAllUnits[0].EMmotorstarter[6].et200SpMotorstarterOutputs[0..1].coldStart := FALSE;
   Et200SpMotorstarterInterfaceAllUnits[0].EMmotorstarter[7].et200SpMotorstarterOutputs[0..1].coldStart := FALSE;
   Et200SpMotorstarterInterfaceAllUnits[0].EMmotorstarter[0].et200SpMotorstarterOutputs[0..1].reserve4 := FALSE;
   Et200SpMotorstarterInterfaceAllUnits[0].EMmotorstarter[1].et200SpMotorstarterOutputs[0..1].reserve4 := FALSE;
   Et200SpMotorstarterInterfaceAllUnits[0].EMmotorstarter[2].et200SpMotorstarterOutputs[0..1].reserve4 := FALSE;
   Et200SpMotorstarterInterfaceAllUnits[0].EMmotorstarter[3].et200SpMotorstarterOutputs[0..1].reserve4 := FALSE;
   Et200SpMotorstarterInterfaceAllUnits[0].EMmotorstarter[4].et200SpMotorstarterOutputs[0..1].reserve4 := FALSE;
   Et200SpMotorstarterInterfaceAllUnits[0].EMmotorstarter[5].et200SpMotorstarterOutputs[0..1].reserve4 := FALSE;
   Et200SpMotorstarterInterfaceAllUnits[0].EMmotorstarter[6].et200SpMotorstarterOutputs[0..1].reserve4 := FALSE;
   Et200SpMotorstarterInterfaceAllUnits[0].EMmotorstarter[7].et200SpMotorstarterOutputs[0..1].reserve4 := FALSE;
   Et200SpMotorstarterInterfaceAllUnits[0].EMmotorstarter[0].et200SpMotorstarterOutputs[0..1].reserve5 := FALSE;
   Et200SpMotorstarterInterfaceAllUnits[0].EMmotorstarter[1].et200SpMotorstarterOutputs[0..1].reserve5 := FALSE;
   Et200SpMotorstarterInterfaceAllUnits[0].EMmotorstarter[2].et200SpMotorstarterOutputs[0..1].reserve5 := FALSE;
   Et200SpMotorstarterInterfaceAllUnits[0].EMmotorstarter[3].et200SpMotorstarterOutputs[0..1].reserve5 := FALSE;
   Et200SpMotorstarterInterfaceAllUnits[0].EMmotorstarter[4].et200SpMotorstarterOutputs[0..1].reserve5 := FALSE;
   Et200SpMotorstarterInterfaceAllUnits[0].EMmotorstarter[5].et200SpMotorstarterOutputs[0..1].reserve5 := FALSE;
   Et200SpMotorstarterInterfaceAllUnits[0].EMmotorstarter[6].et200SpMotorstarterOutputs[0..1].reserve5 := FALSE;
   Et200SpMotorstarterInterfaceAllUnits[0].EMmotorstarter[7].et200SpMotorstarterOutputs[0..1].reserve5 := FALSE;
   Et200SpMotorstarterInterfaceAllUnits[0].EMmotorstarter[0].et200SpMotorstarterOutputs[0..1].reserve6 := FALSE;
   Et200SpMotorstarterInterfaceAllUnits[0].EMmotorstarter[1].et200SpMotorstarterOutputs[0..1].reserve6 := FALSE;
   Et200SpMotorstarterInterfaceAllUnits[0].EMmotorstarter[2].et200SpMotorstarterOutputs[0..1].reserve6 := FALSE;
   Et200SpMotorstarterInterfaceAllUnits[0].EMmotorstarter[3].et200SpMotorstarterOutputs[0..1].reserve6 := FALSE;
   Et200SpMotorstarterInterfaceAllUnits[0].EMmotorstarter[4].et200SpMotorstarterOutputs[0..1].reserve6 := FALSE;
   Et200SpMotorstarterInterfaceAllUnits[0].EMmotorstarter[5].et200SpMotorstarterOutputs[0..1].reserve6 := FALSE;
   Et200SpMotorstarterInterfaceAllUnits[0].EMmotorstarter[6].et200SpMotorstarterOutputs[0..1].reserve6 := FALSE;
   Et200SpMotorstarterInterfaceAllUnits[0].EMmotorstarter[7].et200SpMotorstarterOutputs[0..1].reserve6 := FALSE;
   Et200SpMotorstarterInterfaceAllUnits[0].EMmotorstarter[0].et200SpMotorstarterOutputs[0..1].reserve7 := FALSE;
   Et200SpMotorstarterInterfaceAllUnits[0].EMmotorstarter[1].et200SpMotorstarterOutputs[0..1].reserve7 := FALSE;
   Et200SpMotorstarterInterfaceAllUnits[0].EMmotorstarter[2].et200SpMotorstarterOutputs[0..1].reserve7 := FALSE;
   Et200SpMotorstarterInterfaceAllUnits[0].EMmotorstarter[3].et200SpMotorstarterOutputs[0..1].reserve7 := FALSE;
   Et200SpMotorstarterInterfaceAllUnits[0].EMmotorstarter[4].et200SpMotorstarterOutputs[0..1].reserve7 := FALSE;
   Et200SpMotorstarterInterfaceAllUnits[0].EMmotorstarter[5].et200SpMotorstarterOutputs[0..1].reserve7 := FALSE;
   Et200SpMotorstarterInterfaceAllUnits[0].EMmotorstarter[6].et200SpMotorstarterOutputs[0..1].reserve7 := FALSE;
   Et200SpMotorstarterInterfaceAllUnits[0].EMmotorstarter[7].et200SpMotorstarterOutputs[0..1].reserve7 := FALSE;
   Et200SpMotorstarterInterfaceAllUnits[0].EMmotorstarter[0].et200SpMotorstarterOutputs[0..1].reserve8 := FALSE;
   Et200SpMotorstarterInterfaceAllUnits[0].EMmotorstarter[1].et200SpMotorstarterOutputs[0..1].reserve8 := FALSE;
   Et200SpMotorstarterInterfaceAllUnits[0].EMmotorstarter[2].et200SpMotorstarterOutputs[0..1].reserve8 := FALSE;
   Et200SpMotorstarterInterfaceAllUnits[0].EMmotorstarter[3].et200SpMotorstarterOutputs[0..1].reserve8 := FALSE;
   Et200SpMotorstarterInterfaceAllUnits[0].EMmotorstarter[4].et200SpMotorstarterOutputs[0..1].reserve8 := FALSE;
   Et200SpMotorstarterInterfaceAllUnits[0].EMmotorstarter[5].et200SpMotorstarterOutputs[0..1].reserve8 := FALSE;
   Et200SpMotorstarterInterfaceAllUnits[0].EMmotorstarter[6].et200SpMotorstarterOutputs[0..1].reserve8 := FALSE;
   Et200SpMotorstarterInterfaceAllUnits[0].EMmotorstarter[7].et200SpMotorstarterOutputs[0..1].reserve8 := FALSE;
   Et200SpMotorstarterInterfaceAllUnits[0].EMmotorstarter[0].et200SpMotorstarterOutputs[0..1].reserve9 := FALSE;
   Et200SpMotorstarterInterfaceAllUnits[0].EMmotorstarter[1].et200SpMotorstarterOutputs[0..1].reserve9 := FALSE;
   Et200SpMotorstarterInterfaceAllUnits[0].EMmotorstarter[2].et200SpMotorstarterOutputs[0..1].reserve9 := FALSE;
   Et200SpMotorstarterInterfaceAllUnits[0].EMmotorstarter[3].et200SpMotorstarterOutputs[0..1].reserve9 := FALSE;
   Et200SpMotorstarterInterfaceAllUnits[0].EMmotorstarter[4].et200SpMotorstarterOutputs[0..1].reserve9 := FALSE;
   Et200SpMotorstarterInterfaceAllUnits[0].EMmotorstarter[5].et200SpMotorstarterOutputs[0..1].reserve9 := FALSE;
   Et200SpMotorstarterInterfaceAllUnits[0].EMmotorstarter[6].et200SpMotorstarterOutputs[0..1].reserve9 := FALSE;
   Et200SpMotorstarterInterfaceAllUnits[0].EMmotorstarter[7].et200SpMotorstarterOutputs[0..1].reserve9 := FALSE;
   Et200SpMotorstarterInterfaceAllUnits[0].EMmotorstarter[0].et200SpMotorstarterOutputs[0..1].reserve10 := FALSE;
   Et200SpMotorstarterInterfaceAllUnits[0].EMmotorstarter[1].et200SpMotorstarterOutputs[0..1].reserve10 := FALSE;
   Et200SpMotorstarterInterfaceAllUnits[0].EMmotorstarter[2].et200SpMotorstarterOutputs[0..1].reserve10 := FALSE;
   Et200SpMotorstarterInterfaceAllUnits[0].EMmotorstarter[3].et200SpMotorstarterOutputs[0..1].reserve10 := FALSE;
   Et200SpMotorstarterInterfaceAllUnits[0].EMmotorstarter[4].et200SpMotorstarterOutputs[0..1].reserve10 := FALSE;
   Et200SpMotorstarterInterfaceAllUnits[0].EMmotorstarter[5].et200SpMotorstarterOutputs[0..1].reserve10 := FALSE;
   Et200SpMotorstarterInterfaceAllUnits[0].EMmotorstarter[6].et200SpMotorstarterOutputs[0..1].reserve10 := FALSE;
   Et200SpMotorstarterInterfaceAllUnits[0].EMmotorstarter[7].et200SpMotorstarterOutputs[0..1].reserve10 := FALSE;
   Et200SpMotorstarterInterfaceAllUnits[0].EMmotorstarter[0].et200SpMotorstarterOutputs[0..1].disableQuickStop := FALSE;
   Et200SpMotorstarterInterfaceAllUnits[0].EMmotorstarter[1].et200SpMotorstarterOutputs[0..1].disableQuickStop := FALSE;
   Et200SpMotorstarterInterfaceAllUnits[0].EMmotorstarter[2].et200SpMotorstarterOutputs[0..1].disableQuickStop := FALSE;
   Et200SpMotorstarterInterfaceAllUnits[0].EMmotorstarter[3].et200SpMotorstarterOutputs[0..1].disableQuickStop := FALSE;
   Et200SpMotorstarterInterfaceAllUnits[0].EMmotorstarter[4].et200SpMotorstarterOutputs[0..1].disableQuickStop := FALSE;
   Et200SpMotorstarterInterfaceAllUnits[0].EMmotorstarter[5].et200SpMotorstarterOutputs[0..1].disableQuickStop := FALSE;
   Et200SpMotorstarterInterfaceAllUnits[0].EMmotorstarter[6].et200SpMotorstarterOutputs[0..1].disableQuickStop := FALSE;
   Et200SpMotorstarterInterfaceAllUnits[0].EMmotorstarter[7].et200SpMotorstarterOutputs[0..1].disableQuickStop := FALSE;
END_DATA_BLOCK

DATA_BLOCK "PNDevDiagInterface_X1"   // DB261
// stored: InstanceOfName LAF_typeDevDiagInterface, InstanceOfType UDT
"LAF_typeDevDiagInterface"
   // VAR
   //    globalInfoHmi : "LAF_typeDevDiagGlobal";
   //    devStateHmi { ExternalWritable := 'False'} : Array[0..256] of "LAF_typeDevDiagBasic";
   //    devStateUser { ExternalAccessible := 'False'; ExternalVisible := 'False'; ExternalWritable := 'False'} : Array[0..256] of "LAF_typeDevDiagState";
   // END_VAR
BEGIN
   globalInfoHmi.geoAddressSystem := 0;
   globalInfoHmi.maxDevices := 0;
   globalInfoHmi.maxModuls := 0;
   globalInfoHmi.lowestDevNoConfig := 0;
   globalInfoHmi.highestDevNoConfig := 0;
   globalInfoHmi.numberOfDevices.configured := 0;
   globalInfoHmi.numberOfDevices.notPresent := 0;
   globalInfoHmi.numberOfDevices.deactivated := 0;
   globalInfoHmi.numberOfDevices.faulty := 0;
   globalInfoHmi.numberOfDevices.problem := 0;
   globalInfoHmi.devDiagSummary := FALSE;
   globalInfoHmi.blockBusyAfterNewStart := FALSE;
   globalInfoHmi.manualReadAll := FALSE;
   globalInfoHmi.resetHistoryAll := FALSE;
   devStateHmi[0..256].devNumber := 0;
   devStateHmi[0..256].devName := '';
   devStateHmi[0..256].devStateDezCoded := 0;
   devStateHmi[0..256].devStateBitCoded := 16#0000;
   devStateHmi[0..256].first8CharOfMlfb := '';
   devStateUser[0..256].configured := FALSE;
   devStateUser[0..256].faulty := FALSE;
   devStateUser[0..256].deactivated := FALSE;
   devStateUser[0..256].present := FALSE;
   devStateUser[0..256].problem := FALSE;
   devStateUser[0..256].networkError := FALSE;
   devStateUser[0..256].maintenanceRequired := FALSE;
   devStateUser[0..256].maintenanceDemanded := FALSE;
   devStateUser[0..256].wasFaulty := FALSE;
   devStateUser[0..256].wasProblem := FALSE;
   devStateUser[0..256].modulStateSummary := FALSE;
   devStateUser[0..256].spare11 := FALSE;
   devStateUser[0..256].spare12 := FALSE;
   devStateUser[0..256].spare13 := FALSE;
   devStateUser[0..256].spare14 := FALSE;
   devStateUser[0..256].spare15 := FALSE;
END_DATA_BLOCK

DATA_BLOCK "PNDevDiagInterface_X2"   // DB205
// stored: InstanceOfName LAF_typeDevDiagInterface, InstanceOfType UDT
"LAF_typeDevDiagInterface"
   // VAR
   //    globalInfoHmi : "LAF_typeDevDiagGlobal";
   //    devStateHmi { ExternalWritable := 'False'} : Array[0..256] of "LAF_typeDevDiagBasic";
   //    devStateUser { ExternalAccessible := 'False'; ExternalVisible := 'False'; ExternalWritable := 'False'} : Array[0..256] of "LAF_typeDevDiagState";
   // END_VAR
BEGIN
   globalInfoHmi.geoAddressSystem := 0;
   globalInfoHmi.maxDevices := 0;
   globalInfoHmi.maxModuls := 0;
   globalInfoHmi.lowestDevNoConfig := 0;
   globalInfoHmi.highestDevNoConfig := 0;
   globalInfoHmi.numberOfDevices.configured := 0;
   globalInfoHmi.numberOfDevices.notPresent := 0;
   globalInfoHmi.numberOfDevices.deactivated := 0;
   globalInfoHmi.numberOfDevices.faulty := 0;
   globalInfoHmi.numberOfDevices.problem := 0;
   globalInfoHmi.devDiagSummary := FALSE;
   globalInfoHmi.blockBusyAfterNewStart := FALSE;
   globalInfoHmi.manualReadAll := FALSE;
   globalInfoHmi.resetHistoryAll := FALSE;
   devStateHmi[0..256].devNumber := 0;
   devStateHmi[0..256].devName := '';
   devStateHmi[0..256].devStateDezCoded := 0;
   devStateHmi[0..256].devStateBitCoded := 16#0000;
   devStateHmi[0..256].first8CharOfMlfb := '';
   devStateUser[0..256].configured := FALSE;
   devStateUser[0..256].faulty := FALSE;
   devStateUser[0..256].deactivated := FALSE;
   devStateUser[0..256].present := FALSE;
   devStateUser[0..256].problem := FALSE;
   devStateUser[0..256].networkError := FALSE;
   devStateUser[0..256].maintenanceRequired := FALSE;
   devStateUser[0..256].maintenanceDemanded := FALSE;
   devStateUser[0..256].wasFaulty := FALSE;
   devStateUser[0..256].wasProblem := FALSE;
   devStateUser[0..256].modulStateSummary := FALSE;
   devStateUser[0..256].spare11 := FALSE;
   devStateUser[0..256].spare12 := FALSE;
   devStateUser[0..256].spare13 := FALSE;
   devStateUser[0..256].spare14 := FALSE;
   devStateUser[0..256].spare15 := FALSE;
END_DATA_BLOCK

DATA_BLOCK "PNDevDiagStatus"   // DB231
// stored: InstanceOfName LER_DiagnosticsInterface, InstanceOfType UDT
"LER_DiagnosticsInterface"
   // VAR
   //    DevState { S7_SetPoint := 'True'} : "LER_DevState";
   //    DigState { S7_SetPoint := 'True'} : Array[0..15] of Bool;
   //    Station_Position : Int := 0;
   // END_VAR
BEGIN
   DevState.DevState_X1.staticDevState1[0..100].devNumber := 0;
   DevState.DevState_X1.staticDevState1[0..100].devName := '';
   DevState.DevState_X1.staticDevState1[0..100].devStateDezCoded := 0;
   DevState.DevState_X1.staticDevState1[0..100].devStateBitCoded := 16#0000;
   DevState.DevState_X1.staticDevState1[0..100].first8CharOfMlfb := '';
   DevState.DevState_X1.staticDevState2[0..100].devNumber := 0;
   DevState.DevState_X1.staticDevState2[0..100].devName := '';
   DevState.DevState_X1.staticDevState2[0..100].devStateDezCoded := 0;
   DevState.DevState_X1.staticDevState2[0..100].devStateBitCoded := 16#0000;
   DevState.DevState_X1.staticDevState2[0..100].first8CharOfMlfb := '';
   DevState.DevState_X1.staticDevState3[0..100].devNumber := 0;
   DevState.DevState_X1.staticDevState3[0..100].devName := '';
   DevState.DevState_X1.staticDevState3[0..100].devStateDezCoded := 0;
   DevState.DevState_X1.staticDevState3[0..100].devStateBitCoded := 16#0000;
   DevState.DevState_X1.staticDevState3[0..100].first8CharOfMlfb := '';
   DevState.DevState_X1.staticDevState4[0..100].devNumber := 0;
   DevState.DevState_X1.staticDevState4[0..100].devName := '';
   DevState.DevState_X1.staticDevState4[0..100].devStateDezCoded := 0;
   DevState.DevState_X1.staticDevState4[0..100].devStateBitCoded := 16#0000;
   DevState.DevState_X1.staticDevState4[0..100].first8CharOfMlfb := '';
   DevState.DevState_X1.staticDevState5[0..100].devNumber := 0;
   DevState.DevState_X1.staticDevState5[0..100].devName := '';
   DevState.DevState_X1.staticDevState5[0..100].devStateDezCoded := 0;
   DevState.DevState_X1.staticDevState5[0..100].devStateBitCoded := 16#0000;
   DevState.DevState_X1.staticDevState5[0..100].first8CharOfMlfb := '';
   DevState.DevState_X1.staticDevState6[0..100].devNumber := 0;
   DevState.DevState_X1.staticDevState6[0..100].devName := '';
   DevState.DevState_X1.staticDevState6[0..100].devStateDezCoded := 0;
   DevState.DevState_X1.staticDevState6[0..100].devStateBitCoded := 16#0000;
   DevState.DevState_X1.staticDevState6[0..100].first8CharOfMlfb := '';
   DevState.DevState_X1.staticDevState7[0..100].devNumber := 0;
   DevState.DevState_X1.staticDevState7[0..100].devName := '';
   DevState.DevState_X1.staticDevState7[0..100].devStateDezCoded := 0;
   DevState.DevState_X1.staticDevState7[0..100].devStateBitCoded := 16#0000;
   DevState.DevState_X1.staticDevState7[0..100].first8CharOfMlfb := '';
   DevState.DevState_X1.staticDevState8[0..100].devNumber := 0;
   DevState.DevState_X1.staticDevState8[0..100].devName := '';
   DevState.DevState_X1.staticDevState8[0..100].devStateDezCoded := 0;
   DevState.DevState_X1.staticDevState8[0..100].devStateBitCoded := 16#0000;
   DevState.DevState_X1.staticDevState8[0..100].first8CharOfMlfb := '';
   DevState.DevState_X1.staticDevState9[0..100].devNumber := 0;
   DevState.DevState_X1.staticDevState9[0..100].devName := '';
   DevState.DevState_X1.staticDevState9[0..100].devStateDezCoded := 0;
   DevState.DevState_X1.staticDevState9[0..100].devStateBitCoded := 16#0000;
   DevState.DevState_X1.staticDevState9[0..100].first8CharOfMlfb := '';
   DevState.DevState_X1.staticDevState10[0..100].devNumber := 0;
   DevState.DevState_X1.staticDevState10[0..100].devName := '';
   DevState.DevState_X1.staticDevState10[0..100].devStateDezCoded := 0;
   DevState.DevState_X1.staticDevState10[0..100].devStateBitCoded := 16#0000;
   DevState.DevState_X1.staticDevState10[0..100].first8CharOfMlfb := '';
   DevState.DevState_X1.staticDevState11[0..100].devNumber := 0;
   DevState.DevState_X1.staticDevState11[0..100].devName := '';
   DevState.DevState_X1.staticDevState11[0..100].devStateDezCoded := 0;
   DevState.DevState_X1.staticDevState11[0..100].devStateBitCoded := 16#0000;
   DevState.DevState_X1.staticDevState11[0..100].first8CharOfMlfb := '';
   DevState.DevState_X1.staticDevState12[0..100].devNumber := 0;
   DevState.DevState_X1.staticDevState12[0..100].devName := '';
   DevState.DevState_X1.staticDevState12[0..100].devStateDezCoded := 0;
   DevState.DevState_X1.staticDevState12[0..100].devStateBitCoded := 16#0000;
   DevState.DevState_X1.staticDevState12[0..100].first8CharOfMlfb := '';
   DevState.DevState_X1.staticDevState13[0..100].devNumber := 0;
   DevState.DevState_X1.staticDevState13[0..100].devName := '';
   DevState.DevState_X1.staticDevState13[0..100].devStateDezCoded := 0;
   DevState.DevState_X1.staticDevState13[0..100].devStateBitCoded := 16#0000;
   DevState.DevState_X1.staticDevState13[0..100].first8CharOfMlfb := '';
   DevState.DevState_X1.staticDevState14[0..100].devNumber := 0;
   DevState.DevState_X1.staticDevState14[0..100].devName := '';
   DevState.DevState_X1.staticDevState14[0..100].devStateDezCoded := 0;
   DevState.DevState_X1.staticDevState14[0..100].devStateBitCoded := 16#0000;
   DevState.DevState_X1.staticDevState14[0..100].first8CharOfMlfb := '';
   DevState.DevState_X1.staticDevState15[0..100].devNumber := 0;
   DevState.DevState_X1.staticDevState15[0..100].devName := '';
   DevState.DevState_X1.staticDevState15[0..100].devStateDezCoded := 0;
   DevState.DevState_X1.staticDevState15[0..100].devStateBitCoded := 16#0000;
   DevState.DevState_X1.staticDevState15[0..100].first8CharOfMlfb := '';
   DevState.DevState_X2.staticDevState1[0..100].devNumber := 0;
   DevState.DevState_X2.staticDevState1[0..100].devName := '';
   DevState.DevState_X2.staticDevState1[0..100].devStateDezCoded := 0;
   DevState.DevState_X2.staticDevState1[0..100].devStateBitCoded := 16#0000;
   DevState.DevState_X2.staticDevState1[0..100].first8CharOfMlfb := '';
   DevState.DevState_X2.staticDevState2[0..100].devNumber := 0;
   DevState.DevState_X2.staticDevState2[0..100].devName := '';
   DevState.DevState_X2.staticDevState2[0..100].devStateDezCoded := 0;
   DevState.DevState_X2.staticDevState2[0..100].devStateBitCoded := 16#0000;
   DevState.DevState_X2.staticDevState2[0..100].first8CharOfMlfb := '';
   DevState.DevState_X2.staticDevState3[0..100].devNumber := 0;
   DevState.DevState_X2.staticDevState3[0..100].devName := '';
   DevState.DevState_X2.staticDevState3[0..100].devStateDezCoded := 0;
   DevState.DevState_X2.staticDevState3[0..100].devStateBitCoded := 16#0000;
   DevState.DevState_X2.staticDevState3[0..100].first8CharOfMlfb := '';
   DevState.DevState_X2.staticDevState4[0..100].devNumber := 0;
   DevState.DevState_X2.staticDevState4[0..100].devName := '';
   DevState.DevState_X2.staticDevState4[0..100].devStateDezCoded := 0;
   DevState.DevState_X2.staticDevState4[0..100].devStateBitCoded := 16#0000;
   DevState.DevState_X2.staticDevState4[0..100].first8CharOfMlfb := '';
   DevState.DevState_X2.staticDevState5[0..100].devNumber := 0;
   DevState.DevState_X2.staticDevState5[0..100].devName := '';
   DevState.DevState_X2.staticDevState5[0..100].devStateDezCoded := 0;
   DevState.DevState_X2.staticDevState5[0..100].devStateBitCoded := 16#0000;
   DevState.DevState_X2.staticDevState5[0..100].first8CharOfMlfb := '';
   DevState.DevState_X2.staticDevState6[0..100].devNumber := 0;
   DevState.DevState_X2.staticDevState6[0..100].devName := '';
   DevState.DevState_X2.staticDevState6[0..100].devStateDezCoded := 0;
   DevState.DevState_X2.staticDevState6[0..100].devStateBitCoded := 16#0000;
   DevState.DevState_X2.staticDevState6[0..100].first8CharOfMlfb := '';
   DevState.DevState_X2.staticDevState7[0..100].devNumber := 0;
   DevState.DevState_X2.staticDevState7[0..100].devName := '';
   DevState.DevState_X2.staticDevState7[0..100].devStateDezCoded := 0;
   DevState.DevState_X2.staticDevState7[0..100].devStateBitCoded := 16#0000;
   DevState.DevState_X2.staticDevState7[0..100].first8CharOfMlfb := '';
   DevState.DevState_X2.staticDevState8[0..100].devNumber := 0;
   DevState.DevState_X2.staticDevState8[0..100].devName := '';
   DevState.DevState_X2.staticDevState8[0..100].devStateDezCoded := 0;
   DevState.DevState_X2.staticDevState8[0..100].devStateBitCoded := 16#0000;
   DevState.DevState_X2.staticDevState8[0..100].first8CharOfMlfb := '';
   DevState.DevState_X2.staticDevState9[0..100].devNumber := 0;
   DevState.DevState_X2.staticDevState9[0..100].devName := '';
   DevState.DevState_X2.staticDevState9[0..100].devStateDezCoded := 0;
   DevState.DevState_X2.staticDevState9[0..100].devStateBitCoded := 16#0000;
   DevState.DevState_X2.staticDevState9[0..100].first8CharOfMlfb := '';
   DevState.DevState_X2.staticDevState10[0..100].devNumber := 0;
   DevState.DevState_X2.staticDevState10[0..100].devName := '';
   DevState.DevState_X2.staticDevState10[0..100].devStateDezCoded := 0;
   DevState.DevState_X2.staticDevState10[0..100].devStateBitCoded := 16#0000;
   DevState.DevState_X2.staticDevState10[0..100].first8CharOfMlfb := '';
   DevState.DevState_X2.staticDevState11[0..100].devNumber := 0;
   DevState.DevState_X2.staticDevState11[0..100].devName := '';
   DevState.DevState_X2.staticDevState11[0..100].devStateDezCoded := 0;
   DevState.DevState_X2.staticDevState11[0..100].devStateBitCoded := 16#0000;
   DevState.DevState_X2.staticDevState11[0..100].first8CharOfMlfb := '';
   DevState.DevState_X2.staticDevState12[0..100].devNumber := 0;
   DevState.DevState_X2.staticDevState12[0..100].devName := '';
   DevState.DevState_X2.staticDevState12[0..100].devStateDezCoded := 0;
   DevState.DevState_X2.staticDevState12[0..100].devStateBitCoded := 16#0000;
   DevState.DevState_X2.staticDevState12[0..100].first8CharOfMlfb := '';
   DevState.DevState_X2.staticDevState13[0..100].devNumber := 0;
   DevState.DevState_X2.staticDevState13[0..100].devName := '';
   DevState.DevState_X2.staticDevState13[0..100].devStateDezCoded := 0;
   DevState.DevState_X2.staticDevState13[0..100].devStateBitCoded := 16#0000;
   DevState.DevState_X2.staticDevState13[0..100].first8CharOfMlfb := '';
   DevState.DevState_X2.staticDevState14[0..100].devNumber := 0;
   DevState.DevState_X2.staticDevState14[0..100].devName := '';
   DevState.DevState_X2.staticDevState14[0..100].devStateDezCoded := 0;
   DevState.DevState_X2.staticDevState14[0..100].devStateBitCoded := 16#0000;
   DevState.DevState_X2.staticDevState14[0..100].first8CharOfMlfb := '';
   DevState.DevState_X2.staticDevState15[0..100].devNumber := 0;
   DevState.DevState_X2.staticDevState15[0..100].devName := '';
   DevState.DevState_X2.staticDevState15[0..100].devStateDezCoded := 0;
   DevState.DevState_X2.staticDevState15[0..100].devStateBitCoded := 16#0000;
   DevState.DevState_X2.staticDevState15[0..100].first8CharOfMlfb := '';
   DevState.DevState.staticDevState1[0..100].devNumber := 0;
   DevState.DevState.staticDevState1[0..100].devName := '';
   DevState.DevState.staticDevState1[0..100].devStateDezCoded := 0;
   DevState.DevState.staticDevState1[0..100].devStateBitCoded := 16#0000;
   DevState.DevState.staticDevState1[0..100].first8CharOfMlfb := '';
   DevState.DevState.staticDevState2[0..100].devNumber := 0;
   DevState.DevState.staticDevState2[0..100].devName := '';
   DevState.DevState.staticDevState2[0..100].devStateDezCoded := 0;
   DevState.DevState.staticDevState2[0..100].devStateBitCoded := 16#0000;
   DevState.DevState.staticDevState2[0..100].first8CharOfMlfb := '';
   DevState.DevState.staticDevState3[0..100].devNumber := 0;
   DevState.DevState.staticDevState3[0..100].devName := '';
   DevState.DevState.staticDevState3[0..100].devStateDezCoded := 0;
   DevState.DevState.staticDevState3[0..100].devStateBitCoded := 16#0000;
   DevState.DevState.staticDevState3[0..100].first8CharOfMlfb := '';
   DevState.DevState.staticDevState4[0..100].devNumber := 0;
   DevState.DevState.staticDevState4[0..100].devName := '';
   DevState.DevState.staticDevState4[0..100].devStateDezCoded := 0;
   DevState.DevState.staticDevState4[0..100].devStateBitCoded := 16#0000;
   DevState.DevState.staticDevState4[0..100].first8CharOfMlfb := '';
   DevState.DevState.staticDevState5[0..100].devNumber := 0;
   DevState.DevState.staticDevState5[0..100].devName := '';
   DevState.DevState.staticDevState5[0..100].devStateDezCoded := 0;
   DevState.DevState.staticDevState5[0..100].devStateBitCoded := 16#0000;
   DevState.DevState.staticDevState5[0..100].first8CharOfMlfb := '';
   DevState.DevState.staticDevState6[0..100].devNumber := 0;
   DevState.DevState.staticDevState6[0..100].devName := '';
   DevState.DevState.staticDevState6[0..100].devStateDezCoded := 0;
   DevState.DevState.staticDevState6[0..100].devStateBitCoded := 16#0000;
   DevState.DevState.staticDevState6[0..100].first8CharOfMlfb := '';
   DevState.DevState.staticDevState7[0..100].devNumber := 0;
   DevState.DevState.staticDevState7[0..100].devName := '';
   DevState.DevState.staticDevState7[0..100].devStateDezCoded := 0;
   DevState.DevState.staticDevState7[0..100].devStateBitCoded := 16#0000;
   DevState.DevState.staticDevState7[0..100].first8CharOfMlfb := '';
   DevState.DevState.staticDevState8[0..100].devNumber := 0;
   DevState.DevState.staticDevState8[0..100].devName := '';
   DevState.DevState.staticDevState8[0..100].devStateDezCoded := 0;
   DevState.DevState.staticDevState8[0..100].devStateBitCoded := 16#0000;
   DevState.DevState.staticDevState8[0..100].first8CharOfMlfb := '';
   DevState.DevState.staticDevState9[0..100].devNumber := 0;
   DevState.DevState.staticDevState9[0..100].devName := '';
   DevState.DevState.staticDevState9[0..100].devStateDezCoded := 0;
   DevState.DevState.staticDevState9[0..100].devStateBitCoded := 16#0000;
   DevState.DevState.staticDevState9[0..100].first8CharOfMlfb := '';
   DevState.DevState.staticDevState10[0..100].devNumber := 0;
   DevState.DevState.staticDevState10[0..100].devName := '';
   DevState.DevState.staticDevState10[0..100].devStateDezCoded := 0;
   DevState.DevState.staticDevState10[0..100].devStateBitCoded := 16#0000;
   DevState.DevState.staticDevState10[0..100].first8CharOfMlfb := '';
   DevState.DevState.staticDevState11[0..100].devNumber := 0;
   DevState.DevState.staticDevState11[0..100].devName := '';
   DevState.DevState.staticDevState11[0..100].devStateDezCoded := 0;
   DevState.DevState.staticDevState11[0..100].devStateBitCoded := 16#0000;
   DevState.DevState.staticDevState11[0..100].first8CharOfMlfb := '';
   DevState.DevState.staticDevState12[0..100].devNumber := 0;
   DevState.DevState.staticDevState12[0..100].devName := '';
   DevState.DevState.staticDevState12[0..100].devStateDezCoded := 0;
   DevState.DevState.staticDevState12[0..100].devStateBitCoded := 16#0000;
   DevState.DevState.staticDevState12[0..100].first8CharOfMlfb := '';
   DevState.DevState.staticDevState13[0..100].devNumber := 0;
   DevState.DevState.staticDevState13[0..100].devName := '';
   DevState.DevState.staticDevState13[0..100].devStateDezCoded := 0;
   DevState.DevState.staticDevState13[0..100].devStateBitCoded := 16#0000;
   DevState.DevState.staticDevState13[0..100].first8CharOfMlfb := '';
   DevState.DevState.staticDevState14[0..100].devNumber := 0;
   DevState.DevState.staticDevState14[0..100].devName := '';
   DevState.DevState.staticDevState14[0..100].devStateDezCoded := 0;
   DevState.DevState.staticDevState14[0..100].devStateBitCoded := 16#0000;
   DevState.DevState.staticDevState14[0..100].first8CharOfMlfb := '';
   DevState.DevState.staticDevState15[0..100].devNumber := 0;
   DevState.DevState.staticDevState15[0..100].devName := '';
   DevState.DevState.staticDevState15[0..100].devStateDezCoded := 0;
   DevState.DevState.staticDevState15[0..100].devStateBitCoded := 16#0000;
   DevState.DevState.staticDevState15[0..100].first8CharOfMlfb := '';
   DigState[0] := FALSE;
   DigState[1..9] := TRUE;
   DigState[10..15] := FALSE;
END_DATA_BLOCK

DATA_BLOCK "InstCompValEqOr1"   // DB132
TITLE = Instanz CompValEqOr1 / Instance CompValEqOr1
{ DB_Accessible_From_OPC_UA := 'FALSE' }
AUTHOR : SICAR
FAMILY : Miscellaneous
VERSION : 1.0
// Instanz DB / Instance DB
// stored: DBAccessibleFromOPCUA false, InstanceOfName CompValEqOr, InstanceOfType FB
"CompValEqOr"
BEGIN
END_DATA_BLOCK

DATA_BLOCK "InstCompValEqOr2"   // DB133
TITLE = Instanz CompValEqOr2 / Instance CompValEqOr2
{ DB_Accessible_From_OPC_UA := 'FALSE' }
AUTHOR : SICAR
FAMILY : Miscellaneous
VERSION : 1.0
// Instanz DB / Instance DB
// stored: DBAccessibleFromOPCUA false, InstanceOfName CompValEqOr, InstanceOfType FB
"CompValEqOr"
BEGIN
END_DATA_BLOCK

DATA_BLOCK "InstCounterDataset1"   // DB65
TITLE = Instanz CounterDataset1 / Instance CounterDataset1
{ DB_Accessible_From_OPC_UA := 'FALSE' }
AUTHOR : SICAR
FAMILY : ProdData
// Instanz DB / Instance DB
// stored: DBAccessibleFromOPCUA false, InstanceOfName LSicar_ProdDataCounter, InstanceOfType FB
"LSicar_ProdDataCounter"
   // VAR_INPUT
   //    numberConfigDataSets { ExternalAccessible := 'False'; ExternalVisible := 'False'; ExternalWritable := 'False'} : Int := 0;
   //    dataSetNumber { ExternalAccessible := 'False'; ExternalVisible := 'False'; ExternalWritable := 'False'} : UInt := 0;
   // END_VAR
   // VAR_IN_OUT
   //    numberOfDataSets : "LSicar_typeNumberOfDataSets";
   //    dataSet : "LSicar_typeCounter";
   // END_VAR
   // VAR
   //    statCounter { ExternalAccessible := 'False'; ExternalVisible := 'False'; ExternalWritable := 'False'} : Array[0..20] of "LSicar_typeEdgePulseStruct";
   //    statRisEdgeResetAllExt { ExternalAccessible := 'False'; ExternalVisible := 'False'; ExternalWritable := 'False'} : Bool := FALSE;
   //    statPosPulseResetAllExt { ExternalAccessible := 'False'; ExternalVisible := 'False'; ExternalWritable := 'False'} : Bool := FALSE;
   //    statRisEdgeResetAll { ExternalAccessible := 'False'; ExternalVisible := 'False'; ExternalWritable := 'False'} : Bool := FALSE;
   //    statPosPulseResetAll { ExternalAccessible := 'False'; ExternalVisible := 'False'; ExternalWritable := 'False'} : Bool := FALSE;
   // END_VAR
BEGIN
   statCounter[0..20].risEdgeCountUp := FALSE;
   statCounter[0..20].posPulseCountUp := FALSE;
   statCounter[0..20].risEdgeCountDown := FALSE;
   statCounter[0..20].posPulseCountDown := FALSE;
   statCounter[0..20].risEdgeReset := FALSE;
   statCounter[0..20].posPulseReset := FALSE;
END_DATA_BLOCK

DATA_BLOCK "InstCounterDataset2"   // DB66
TITLE = Instanz CounterDataSet2 / Instance CounterDataSet2
{ DB_Accessible_From_OPC_UA := 'FALSE' }
AUTHOR : SICAR
FAMILY : ProdData
// Instanz DB / Instance DB
// stored: DBAccessibleFromOPCUA false, InstanceOfName LSicar_ProdDataCounter, InstanceOfType FB
"LSicar_ProdDataCounter"
   // VAR_INPUT
   //    numberConfigDataSets { ExternalAccessible := 'False'; ExternalVisible := 'False'; ExternalWritable := 'False'} : Int := 0;
   //    dataSetNumber { ExternalAccessible := 'False'; ExternalVisible := 'False'; ExternalWritable := 'False'} : UInt := 0;
   // END_VAR
   // VAR_IN_OUT
   //    numberOfDataSets : "LSicar_typeNumberOfDataSets";
   //    dataSet : "LSicar_typeCounter";
   // END_VAR
   // VAR
   //    statCounter { ExternalAccessible := 'False'; ExternalVisible := 'False'; ExternalWritable := 'False'} : Array[0..20] of "LSicar_typeEdgePulseStruct";
   //    statRisEdgeResetAllExt { ExternalAccessible := 'False'; ExternalVisible := 'False'; ExternalWritable := 'False'} : Bool := FALSE;
   //    statPosPulseResetAllExt { ExternalAccessible := 'False'; ExternalVisible := 'False'; ExternalWritable := 'False'} : Bool := FALSE;
   //    statRisEdgeResetAll { ExternalAccessible := 'False'; ExternalVisible := 'False'; ExternalWritable := 'False'} : Bool := FALSE;
   //    statPosPulseResetAll { ExternalAccessible := 'False'; ExternalVisible := 'False'; ExternalWritable := 'False'} : Bool := FALSE;
   // END_VAR
BEGIN
   statCounter[0..20].risEdgeCountUp := FALSE;
   statCounter[0..20].posPulseCountUp := FALSE;
   statCounter[0..20].risEdgeCountDown := FALSE;
   statCounter[0..20].posPulseCountDown := FALSE;
   statCounter[0..20].risEdgeReset := FALSE;
   statCounter[0..20].posPulseReset := FALSE;
END_DATA_BLOCK

